LIN {X 0,Y 260.997,Z 552.106,A -85,B 0,C 180,E1 -19941.733,E2 -19941.733} C_VEL
LIN {X 0,Y 261.38,Z 553.874,A -85,B 0,C 180,E1 -19943.77,E2 -19943.77} C_VEL
LIN {X 0,Y 261.439,Z 557.559,A -85,B 0,C 180,E1 -19946.444,E2 -19946.444} C_VEL
LIN {X 0,Y 260.966,Z 561.356,A -85,B 0,C 180,E1 -19948.526,E2 -19948.526} C_VEL
LIN {X 0,Y 260.147,Z 563.053,A -85,B 0,C 180,E1 -19949.117,E2 -19949.117} C_VEL
LIN {X 0,Y 253.93,Z 571.512,A -85,B 0,C 180,E1 -19951.483,E2 -19951.483} C_VEL
LIN {X 0,Y 248.241,Z 578.441,A -85,B 0,C 180,E1 -19953.971,E2 -19953.971} C_VEL
LIN {X 0,Y 243.866,Z 583.268,A -85,B 0,C 180,E1 -19956.205,E2 -19956.205} C_VEL
LIN {X 0,Y 238.865,Z 588.279,A -85,B 0,C 180,E1 -19959.325,E2 -19959.325} C_VEL
LIN {X 0,Y 234.733,Z 591.746,A -85,B 0,C 180,E1 -19962.578,E2 -19962.578} C_VEL
LIN {X 0,Y 232.898,Z 592.963,A -85,B 0,C 180,E1 -19964.242,E2 -19964.242} C_VEL
LIN {X 0,Y 230.123,Z 594.324,A -85,B 0,C 180,E1 -19967.656,E2 -19967.656} C_VEL
LIN {X 0,Y 227.905,Z 594.264,A -85,B 0,C 180,E1 -19971.131,E2 -19971.131} C_VEL
LIN {X 0,Y 226.815,Z 592.766,A -85,B 0,C 180,E1 -19974.667,E2 -19974.667} C_VEL
LIN {X 0,Y 226.415,Z 591.482,A -85,B 0,C 180,E1 -19976.441,E2 -19976.441} C_VEL
LIN {X 0,Y 225.975,Z 587.71,A -85,B 0,C 180,E1 -19980,E2 -19980} C_VEL
LIN {X 0,Y 226.019,Z 583.819,A -85,B 0,C 180,E1 -19982.674,E2 -19982.674} C_VEL
LIN {X 0,Y 226.077,Z 578.823,A -85,B 0,C 180,E1 -19985.352,E2 -19985.352} C_VEL
LIN {X 0,Y 226.623,Z 571.523,A -85,B 0,C 180,E1 -19988.471,E2 -19988.471} C_VEL
LIN {X 0,Y 227.3,Z 563.747,A -85,B 0,C 180,E1 -19991.143,E2 -19991.143} C_VEL
LIN {X 0,Y 228.271,Z 554.253,A -85,B 0,C 180,E1 -19993.805,E2 -19993.805} C_VEL
LIN {X 0,Y 229.552,Z 543.626,A -85,B 0,C 180,E1 -19996.223,E2 -19996.223} C_VEL
LIN {X 0,Y 230.932,Z 531.732,A -85,B 0,C 180,E1 -19998.406,E2 -19998.406} C_VEL
LIN {X 0,Y 232.043,Z 520.197,A -85,B 0,C 180,E1 -20000.13,E2 -20000.13} C_VEL
LIN {X 0,Y 229.504,Z 506.12,A -85,B 0,C 180,E1 -20001.897,E2 -20001.897} C_VEL
LIN {X 0,Y 227.192,Z 492.741,A -85,B 0,C 180,E1 -20003.213,E2 -20003.213} C_VEL
LIN {X 0,Y 226.512,Z 488.275,A -85,B 0,C 180,E1 -20003.585,E2 -20003.585} C_VEL
LIN {X 0,Y 226.901,Z 488.225,A -85,B 0,C 180,E1 -20007.685,E2 -20007.685} C_VEL
LIN {X 0,Y 227.309,Z 488.167,A -85,B 0,C 180,E1 -20011.71,E2 -20011.71} C_VEL
LIN {X 0,Y 227.697,Z 488.121,A -85,B 0,C 180,E1 -20015.906,E2 -20015.906} C_VEL
LIN {X 0,Y 227.817,Z 488.105,A -85,B 0,C 180,E1 -20019.535,E2 -20019.535} C_VEL
LIN {X 0,Y 227.812,Z 488.105,A -85,B 0,C 180,E1 -20022.743,E2 -20022.743} C_VEL
LIN {X 0,Y 227.817,Z 488.105,A -85,B 0,C 180,E1 -20027.259,E2 -20027.259} C_VEL
LIN {X 0,Y 227.873,Z 488.098,A -85,B 0,C 180,E1 -20031.914,E2 -20031.914} C_VEL
LIN {X 0,Y 227.895,Z 488.097,A -85,B 0,C 180,E1 -20036.373,E2 -20036.373} C_VEL
LIN {X 0,Y 227.922,Z 488.093,A -85,B 0,C 180,E1 -20040.438,E2 -20040.438} C_VEL
LIN {X 0,Y 227.933,Z 488.092,A -85,B 0,C 180,E1 -20044.426,E2 -20044.426} C_VEL
LIN {X 0,Y 227.966,Z 488.087,A -85,B 0,C 180,E1 -20048.287,E2 -20048.287} C_VEL
LIN {X 0,Y 228.039,Z 488.078,A -85,B 0,C 180,E1 -20052.826,E2 -20052.826} C_VEL
LIN {X 0,Y 228.099,Z 488.068,A -85,B 0,C 180,E1 -20057.545,E2 -20057.545} C_VEL
LIN {X 0,Y 228.33,Z 488.041,A -85,B 0,C 180,E1 -20061.147,E2 -20061.147} C_VEL
LIN {X 0,Y 228.363,Z 488.036,A -85,B 0,C 180,E1 -20062.929,E2 -20062.929} C_VEL
LIN {X 0,Y 228.559,Z 488.015,A -85,B 0,C 180,E1 -20068.238,E2 -20068.238} C_VEL
LIN {X 0,Y 228.558,Z 488.015,A -85,B 0,C 180,E1 -20071.762,E2 -20071.762} C_VEL
LIN {X 0,Y 228.316,Z 488.042,A -85,B 0,C 180,E1 -20077.073,E2 -20077.073} C_VEL
LIN {X 0,Y 228.15,Z 488.063,A -85,B 0,C 180,E1 -20080.651,E2 -20080.651} C_VEL
LIN {X 0,Y 228.07,Z 488.074,A -85,B 0,C 180,E1 -20084.272,E2 -20084.272} C_VEL
LIN {X 0,Y 228.007,Z 488.085,A -85,B 0,C 180,E1 -20087.953,E2 -20087.953} C_VEL
LIN {X 0,Y 227.934,Z 488.089,A -85,B 0,C 180,E1 -20092.329,E2 -20092.329} C_VEL
LIN {X 0,Y 227.947,Z 488.089,A -85,B 0,C 180,E1 -20096.602,E2 -20096.602} C_VEL
LIN {X 0,Y 227.912,Z 488.091,A -85,B 0,C 180,E1 -20100.296,E2 -20100.296} C_VEL
LIN {X 0,Y 227.894,Z 488.098,A -85,B 0,C 180,E1 -20103.718,E2 -20103.718} C_VEL
LIN {X 0,Y 227.873,Z 488.098,A -85,B 0,C 180,E1 -20108.086,E2 -20108.086} C_VEL
LIN {X 0,Y 227.817,Z 488.105,A -85,B 0,C 180,E1 -20112.741,E2 -20112.741} C_VEL
LIN {X 0,Y 227.814,Z 488.105,A -85,B 0,C 180,E1 -20117.257,E2 -20117.257} C_VEL
LIN {X 0,Y 227.826,Z 488.107,A -85,B 0,C 180,E1 -20121.905,E2 -20121.905} C_VEL
LIN {X 0,Y 227.775,Z 488.111,A -85,B 0,C 180,E1 -20124.108,E2 -20124.108} C_VEL
LIN {X 0,Y 227.441,Z 488.151,A -85,B 0,C 180,E1 -20128.31,E2 -20128.31} C_VEL
LIN {X 0,Y 226.941,Z 488.214,A -85,B 0,C 180,E1 -20132.32,E2 -20132.32} C_VEL
LIN {X 0,Y 226.511,Z 488.447,A -85,B 0,C 180,E1 -20136.724,E2 -20136.724} C_VEL
LIN {X 0,Y 228.847,Z 502.265,A -85,B 0,C 180,E1 -20137.982,E2 -20137.982} C_VEL
LIN {X 0,Y 231.402,Z 516.968,A -85,B 0,C 180,E1 -20139.723,E2 -20139.723} C_VEL
LIN {X 0,Y 231.9,Z 519.763,A -85,B 0,C 180,E1 -20140.109,E2 -20140.109} C_VEL
LIN {X 0,Y 230.711,Z 532.571,A -85,B 0,C 180,E1 -20142.035,E2 -20142.035} C_VEL
LIN {X 0,Y 229.325,Z 544.216,A -85,B 0,C 180,E1 -20144.217,E2 -20144.217} C_VEL
LIN {X 0,Y 228.097,Z 554.659,A -85,B 0,C 180,E1 -20146.638,E2 -20146.638} C_VEL
LIN {X 0,Y 227.17,Z 564.012,A -85,B 0,C 180,E1 -20149.302,E2 -20149.302} C_VEL
LIN {X 0,Y 226.478,Z 571.65,A -85,B 0,C 180,E1 -20151.972,E2 -20151.972} C_VEL
LIN {X 0,Y 226.06,Z 577.897,A -85,B 0,C 180,E1 -20154.648,E2 -20154.648} C_VEL
LIN {X 0,Y 226.009,Z 582.973,A -85,B 0,C 180,E1 -20157.326,E2 -20157.326} C_VEL
LIN {X 0,Y 225.947,Z 586.927,A -85,B 0,C 180,E1 -20160,E2 -20160} C_VEL
LIN {X 0,Y 226.391,Z 590.762,A -85,B 0,C 180,E1 -20163.559,E2 -20163.559} C_VEL
LIN {X 0,Y 227.153,Z 593.019,A -85,B 0,C 180,E1 -20167.109,E2 -20167.109} C_VEL
LIN {X 0,Y 228.816,Z 593.825,A -85,B 0,C 180,E1 -20170.619,E2 -20170.619} C_VEL
LIN {X 0,Y 229.985,Z 593.691,A -85,B 0,C 180,E1 -20172.351,E2 -20172.351} C_VEL
LIN {X 0,Y 231.149,Z 593.198,A -85,B 0,C 180,E1 -20174.077,E2 -20174.077} C_VEL
LIN {X 0,Y 234.587,Z 591.116,A -85,B 0,C 180,E1 -20177.433,E2 -20177.433} C_VEL
LIN {X 0,Y 236.432,Z 589.575,A -85,B 0,C 180,E1 -20179.085,E2 -20179.085} C_VEL
LIN {X 0,Y 241.087,Z 585.314,A -85,B 0,C 180,E1 -20182.269,E2 -20182.269} C_VEL
LIN {X 0,Y 246.476,Z 579.492,A -85,B 0,C 180,E1 -20185.322,E2 -20185.322} C_VEL
LIN {X 0,Y 251.935,Z 572.921,A -85,B 0,C 180,E1 -20187.856,E2 -20187.856} C_VEL
LIN {X 0,Y 257.976,Z 564.873,A -85,B 0,C 180,E1 -20190.264,E2 -20190.264} C_VEL
LIN {X 0,Y 261.362,Z 559.796,A -85,B 0,C 180,E1 -20191.544,E2 -20191.544} C_VEL
LIN {X 0,Y 262.125,Z 555.274,A -85,B 0,C 180,E1 -20193.782,E2 -20193.782} C_VEL
LIN {X 0,Y 262.421,Z 551.482,A -85,B 0,C 180,E1 -20196.099,E2 -20196.099} C_VEL
LIN {X 0,Y 262.376,Z 549.202,A -85,B 0,C 180,E1 -20198.03,E2 -20198.03} C_VEL
LIN {X 0,Y 262.053,Z 547.219,A -85,B 0,C 180,E1 -20201.329,E2 -20201.329} C_VEL
LIN {X 0,Y 262.112,Z 546.874,A -85,B 0,C 180,E1 -20204.198,E2 -20204.198} C_VEL
LIN {X 0,Y 262.067,Z 548.078,A -85,B 0,C 180,E1 -20206.392,E2 -20206.392} C_VEL
LIN {X 0,Y 262.09,Z 550.434,A -85,B 0,C 180,E1 -20208.662,E2 -20208.662} C_VEL
LIN {X 0,Y 261.725,Z 553.395,A -85,B 0,C 180,E1 -20210.385,E2 -20210.385} C_VEL
LIN {X 0,Y 261.022,Z 556.614,A -85,B 0,C 180,E1 -20211.737,E2 -20211.737} C_VEL
LIN {X 0,Y 259.769,Z 560.538,A -85,B 0,C 180,E1 -20213.058,E2 -20213.058} C_VEL
LIN {X 0,Y 258.835,Z 562.899,A -85,B 0,C 180,E1 -20213.731,E2 -20213.731} C_VEL
LIN {X 0,Y 256.688,Z 566.806,A -85,B 0,C 180,E1 -20214.61,E2 -20214.61} C_VEL
LIN {X 0,Y 250.235,Z 576.094,A -85,B 0,C 180,E1 -20216.484,E2 -20216.484} C_VEL
LIN {X 0,Y 247.787,Z 579.695,A -85,B 0,C 180,E1 -20217.424,E2 -20217.424} C_VEL
LIN {X 0,Y 247.137,Z 580.788,A -85,B 0,C 180,E1 -20217.775,E2 -20217.775} C_VEL
LIN {X 0,Y 242.575,Z 587.784,A -85,B 0,C 180,E1 -20220.015,E2 -20220.015} C_VEL
LIN {X 0,Y 236.889,Z 595.016,A -85,B 0,C 180,E1 -20222.622,E2 -20222.622} C_VEL
LIN {X 0,Y 231.389,Z 601.575,A -85,B 0,C 180,E1 -20225.697,E2 -20225.697} C_VEL
LIN {X 0,Y 227.708,Z 605.755,A -85,B 0,C 180,E1 -20228.262,E2 -20228.262} C_VEL
LIN {X 0,Y 224.049,Z 609.838,A -85,B 0,C 180,E1 -20231.719,E2 -20231.719} C_VEL
LIN {X 0,Y 221.143,Z 612.568,A -85,B 0,C 180,E1 -20235.271,E2 -20235.271} C_VEL
LIN {X 0,Y 219.574,Z 613.972,A -85,B 0,C 180,E1 -20238.928,E2 -20238.928} C_VEL
LIN {X 0,Y 218.936,Z 613.961,A -85,B 0,C 180,E1 -20242.623,E2 -20242.623} C_VEL
LIN {X 0,Y 218.988,Z 612.5,A -85,B 0,C 180,E1 -20246.32,E2 -20246.32} C_VEL
LIN {X 0,Y 219.639,Z 610.27,A -85,B 0,C 180,E1 -20249.312,E2 -20249.312} C_VEL
LIN {X 0,Y 219.273,Z 612.678,A -85,B 0,C 180,E1 -20251.837,E2 -20251.837} C_VEL
LIN {X 0,Y 218.885,Z 614.828,A -85,B 0,C 180,E1 -20255.528,E2 -20255.528} C_VEL
LIN {X 0,Y 219.122,Z 615.516,A -85,B 0,C 180,E1 -20259.228,E2 -20259.228} C_VEL
LIN {X 0,Y 220.226,Z 614.78,A -85,B 0,C 180,E1 -20262.908,E2 -20262.908} C_VEL
LIN {X 0,Y 222.43,Z 612.714,A -85,B 0,C 180,E1 -20266.521,E2 -20266.521} C_VEL
LIN {X 0,Y 225.697,Z 609.304,A -85,B 0,C 180,E1 -20270.031,E2 -20270.031} C_VEL
LIN {X 0,Y 228.769,Z 605.775,A -85,B 0,C 180,E1 -20272.65,E2 -20272.65} C_VEL
LIN {X 0,Y 233.83,Z 599.998,A -85,B 0,C 180,E1 -20275.837,E2 -20275.837} C_VEL
LIN {X 0,Y 239.21,Z 593.581,A -85,B 0,C 180,E1 -20278.518,E2 -20278.518} C_VEL
LIN {X 0,Y 245.963,Z 584.688,A -85,B 0,C 180,E1 -20281.431,E2 -20281.431} C_VEL
LIN {X 0,Y 248.001,Z 581.154,A -85,B 0,C 180,E1 -20282.577,E2 -20282.577} C_VEL
LIN {X 0,Y 250.573,Z 575.348,A -85,B 0,C 180,E1 -20284.659,E2 -20284.659} C_VEL
LIN {X 0,Y 252.859,Z 568.813,A -85,B 0,C 180,E1 -20287.194,E2 -20287.194} C_VEL
LIN {X 0,Y 254.372,Z 563.772,A -85,B 0,C 180,E1 -20289.455,E2 -20289.455} C_VEL
LIN {X 0,Y 255.197,Z 560.413,A -85,B 0,C 180,E1 -20291.372,E2 -20291.372} C_VEL
LIN {X 0,Y 255.721,Z 557.205,A -85,B 0,C 180,E1 -20294.393,E2 -20294.393} C_VEL
LIN {X 0,Y 255.885,Z 556.408,A -85,B 0,C 180,E1 -20295.57,E2 -20295.57} C_VEL
LIN {X 0,Y 255.914,Z 556.069,A -85,B 0,C 180,E1 -20297.858,E2 -20297.858} C_VEL
LIN {X 0,Y 256.096,Z 556.949,A -85,B 0,C 180,E1 -20300.863,E2 -20300.863} C_VEL
LIN {X 0,Y 256.423,Z 559.105,A -85,B 0,C 180,E1 -20303.785,E2 -20303.785} C_VEL
LIN {X 0,Y 256.219,Z 561.054,A -85,B 0,C 180,E1 -20305.375,E2 -20305.375} C_VEL
LIN {X 0,Y 255.687,Z 564.505,A -85,B 0,C 180,E1 -20307.604,E2 -20307.604} C_VEL
LIN {X 0,Y 254.559,Z 566.477,A -85,B 0,C 180,E1 -20308.362,E2 -20308.362} C_VEL
LIN {X 0,Y 248.996,Z 573.361,A -85,B 0,C 180,E1 -20310.4,E2 -20310.4} C_VEL
LIN {X 0,Y 242.182,Z 580.837,A -85,B 0,C 180,E1 -20313.269,E2 -20313.269} C_VEL
LIN {X 0,Y 237.648,Z 585.3,A -85,B 0,C 180,E1 -20315.542,E2 -20315.542} C_VEL
LIN {X 0,Y 232.423,Z 589.852,A -85,B 0,C 180,E1 -20318.725,E2 -20318.725} C_VEL
LIN {X 0,Y 228.076,Z 592.969,A -85,B 0,C 180,E1 -20322.053,E2 -20322.053} C_VEL
LIN {X 0,Y 226.163,Z 594.008,A -85,B 0,C 180,E1 -20323.76,E2 -20323.76} C_VEL
LIN {X 0,Y 223.23,Z 595.007,A -85,B 0,C 180,E1 -20327.269,E2 -20327.269} C_VEL
LIN {X 0,Y 220.918,Z 594.665,A -85,B 0,C 180,E1 -20330.848,E2 -20330.848} C_VEL
LIN {X 0,Y 219.753,Z 592.868,A -85,B 0,C 180,E1 -20334.495,E2 -20334.495} C_VEL
LIN {X 0,Y 219.051,Z 589.599,A -85,B 0,C 180,E1 -20338.162,E2 -20338.162} C_VEL
LIN {X 0,Y 218.882,Z 586.103,A -85,B 0,C 180,E1 -20340.92,E2 -20340.92} C_VEL
LIN {X 0,Y 218.927,Z 581.625,A -85,B 0,C 180,E1 -20343.682,E2 -20343.682} C_VEL
LIN {X 0,Y 219.255,Z 575.022,A -85,B 0,C 180,E1 -20346.904,E2 -20346.904} C_VEL
LIN {X 0,Y 219.77,Z 567.895,A -85,B 0,C 180,E1 -20349.666,E2 -20349.666} C_VEL
LIN {X 0,Y 220.638,Z 559.205,A -85,B 0,C 180,E1 -20352.417,E2 -20352.417} C_VEL
LIN {X 0,Y 221.801,Z 548.639,A -85,B 0,C 180,E1 -20355.154,E2 -20355.154} C_VEL
LIN {X 0,Y 223.055,Z 537.863,A -85,B 0,C 180,E1 -20357.418,E2 -20357.418} C_VEL
LIN {X 0,Y 224.214,Z 527.533,A -85,B 0,C 180,E1 -20359.216,E2 -20359.216} C_VEL
LIN {X 0,Y 224.919,Z 521.594,A -85,B 0,C 180,E1 -20360.104,E2 -20360.104} C_VEL
LIN {X 0,Y 223.269,Z 511.586,A -85,B 0,C 180,E1 -20361.465,E2 -20361.465} C_VEL
LIN {X 0,Y 220.895,Z 498.112,A -85,B 0,C 180,E1 -20362.962,E2 -20362.962} C_VEL
LIN {X 0,Y 219.504,Z 489.148,A -85,B 0,C 180,E1 -20363.777,E2 -20363.777} C_VEL
LIN {X 0,Y 219.95,Z 489.087,A -85,B 0,C 180,E1 -20368.64,E2 -20368.64} C_VEL
LIN {X 0,Y 220.361,Z 489.032,A -85,B 0,C 180,E1 -20372.833,E2 -20372.833} C_VEL
LIN {X 0,Y 220.71,Z 488.99,A -85,B 0,C 180,E1 -20377.243,E2 -20377.243} C_VEL
LIN {X 0,Y 220.776,Z 488.984,A -85,B 0,C 180,E1 -20380.182,E2 -20380.182} C_VEL
LIN {X 0,Y 220.776,Z 488.985,A -85,B 0,C 180,E1 -20384.454,E2 -20384.454} C_VEL
LIN {X 0,Y 220.778,Z 488.984,A -85,B 0,C 180,E1 -20388.049,E2 -20388.049} C_VEL
LIN {X 0,Y 220.835,Z 488.975,A -85,B 0,C 180,E1 -20392.795,E2 -20392.795} C_VEL
LIN {X 0,Y 220.828,Z 488.975,A -85,B 0,C 180,E1 -20397.246,E2 -20397.246} C_VEL
LIN {X 0,Y 220.84,Z 488.973,A -85,B 0,C 180,E1 -20401.487,E2 -20401.487} C_VEL
LIN {X 0,Y 220.871,Z 488.971,A -85,B 0,C 180,E1 -20405.565,E2 -20405.565} C_VEL
LIN {X 0,Y 220.897,Z 488.965,A -85,B 0,C 180,E1 -20409.514,E2 -20409.514} C_VEL
LIN {X 0,Y 221.021,Z 488.952,A -85,B 0,C 180,E1 -20413.37,E2 -20413.37} C_VEL
LIN {X 0,Y 221.121,Z 488.938,A -85,B 0,C 180,E1 -20419.006,E2 -20419.006} C_VEL
LIN {X 0,Y 221.316,Z 488.915,A -85,B 0,C 180,E1 -20422.702,E2 -20422.702} C_VEL
LIN {X 0,Y 221.517,Z 488.893,A -85,B 0,C 180,E1 -20428.182,E2 -20428.182} C_VEL
LIN {X 0,Y 221.516,Z 488.893,A -85,B 0,C 180,E1 -20431.818,E2 -20431.818} C_VEL
LIN {X 0,Y 221.252,Z 488.923,A -85,B 0,C 180,E1 -20437.3,E2 -20437.3} C_VEL
LIN {X 0,Y 221.086,Z 488.943,A -85,B 0,C 180,E1 -20440.996,E2 -20440.996} C_VEL
LIN {X 0,Y 221.021,Z 488.952,A -85,B 0,C 180,E1 -20446.63,E2 -20446.63} C_VEL
LIN {X 0,Y 220.897,Z 488.966,A -85,B 0,C 180,E1 -20450.486,E2 -20450.486} C_VEL
LIN {X 0,Y 220.871,Z 488.971,A -85,B 0,C 180,E1 -20454.435,E2 -20454.435} C_VEL
LIN {X 0,Y 220.84,Z 488.973,A -85,B 0,C 180,E1 -20458.513,E2 -20458.513} C_VEL
LIN {X 0,Y 220.828,Z 488.975,A -85,B 0,C 180,E1 -20462.754,E2 -20462.754} C_VEL
LIN {X 0,Y 220.842,Z 488.974,A -85,B 0,C 180,E1 -20467.288,E2 -20467.288} C_VEL
LIN {X 0,Y 220.778,Z 488.984,A -85,B 0,C 180,E1 -20471.951,E2 -20471.951} C_VEL
LIN {X 0,Y 220.777,Z 488.985,A -85,B 0,C 180,E1 -20475.546,E2 -20475.546} C_VEL
LIN {X 0,Y 220.79,Z 488.98,A -85,B 0,C 180,E1 -20480.459,E2 -20480.459} C_VEL
LIN {X 0,Y 220.788,Z 488.981,A -85,B 0,C 180,E1 -20482.785,E2 -20482.785} C_VEL
LIN {X 0,Y 220.456,Z 489.02,A -85,B 0,C 180,E1 -20487.183,E2 -20487.183} C_VEL
LIN {X 0,Y 220.268,Z 489.047,A -85,B 0,C 180,E1 -20489.483,E2 -20489.483} C_VEL
LIN {X 0,Y 219.752,Z 489.112,A -85,B 0,C 180,E1 -20493.571,E2 -20493.571} C_VEL
LIN {X 0,Y 219.454,Z 489.149,A -85,B 0,C 180,E1 -20496.505,E2 -20496.505} C_VEL
LIN {X 0,Y 222.105,Z 504.713,A -85,B 0,C 180,E1 -20498.039,E2 -20498.039} C_VEL
LIN {X 0,Y 224.317,Z 517.522,A -85,B 0,C 180,E1 -20499.625,E2 -20499.625} C_VEL
LIN {X 0,Y 224.798,Z 521.395,A -85,B 0,C 180,E1 -20500.176,E2 -20500.176} C_VEL
LIN {X 0,Y 223.456,Z 533.723,A -85,B 0,C 180,E1 -20502.142,E2 -20502.142} C_VEL
LIN {X 0,Y 222.089,Z 545.146,A -85,B 0,C 180,E1 -20504.396,E2 -20504.396} C_VEL
LIN {X 0,Y 220.841,Z 556.293,A -85,B 0,C 180,E1 -20507.128,E2 -20507.128} C_VEL
LIN {X 0,Y 219.895,Z 565.419,A -85,B 0,C 180,E1 -20509.875,E2 -20509.875} C_VEL
LIN {X 0,Y 219.311,Z 572.892,A -85,B 0,C 180,E1 -20512.635,E2 -20512.635} C_VEL
LIN {X 0,Y 218.945,Z 579.457,A -85,B 0,C 180,E1 -20515.643,E2 -20515.643} C_VEL
LIN {X 0,Y 218.9,Z 583.873,A -85,B 0,C 180,E1 -20518.16,E2 -20518.16} C_VEL
LIN {X 0,Y 218.918,Z 587.74,A -85,B 0,C 180,E1 -20520.919,E2 -20520.919} C_VEL
LIN {X 0,Y 219.332,Z 590.677,A -85,B 0,C 180,E1 -20523.674,E2 -20523.674} C_VEL
LIN {X 0,Y 220.113,Z 593.248,A -85,B 0,C 180,E1 -20527.337,E2 -20527.337} C_VEL
LIN {X 0,Y 221.875,Z 594.342,A -85,B 0,C 180,E1 -20530.955,E2 -20530.955} C_VEL
LIN {X 0,Y 224.34,Z 594.036,A -85,B 0,C 180,E1 -20534.514,E2 -20534.514} C_VEL
LIN {X 0,Y 225.965,Z 593.365,A -85,B 0,C 180,E1 -20536.255,E2 -20536.255} C_VEL
LIN {X 0,Y 229.887,Z 590.951,A -85,B 0,C 180,E1 -20539.65,E2 -20539.65} C_VEL
LIN {X 0,Y 234.75,Z 587.071,A -85,B 0,C 180,E1 -20542.904,E2 -20542.904} C_VEL
LIN {X 0,Y 238.859,Z 583.221,A -85,B 0,C 180,E1 -20545.254,E2 -20545.254} C_VEL
LIN {X 0,Y 245.201,Z 576.599,A -85,B 0,C 180,E1 -20548.224,E2 -20548.224} C_VEL
LIN {X 0,Y 251.402,Z 569.264,A -85,B 0,C 180,E1 -20550.676,E2 -20550.676} C_VEL
LIN {X 0,Y 256.107,Z 563.154,A -85,B 0,C 180,E1 -20552.351,E2 -20552.351} C_VEL
LIN {X 0,Y 256.842,Z 560.292,A -85,B 0,C 180,E1 -20553.879,E2 -20553.879} C_VEL
LIN {X 0,Y 257.63,Z 555.851,A -85,B 0,C 180,E1 -20556.88,E2 -20556.88} C_VEL
LIN {X 0,Y 257.614,Z 554.045,A -85,B 0,C 180,E1 -20558.863,E2 -20558.863} C_VEL
LIN {X 0,Y 257.573,Z 552.939,A -85,B 0,C 180,E1 -20560.908,E2 -20560.908} C_VEL
LIN {X 0,Y 257.643,Z 552.453,A -85,B 0,C 180,E1 -20562.996,E2 -20562.996} C_VEL
LIN {X 0,Y 257.679,Z 552.943,A -85,B 0,C 180,E1 -20565.164,E2 -20565.164} C_VEL
LIN {X 0,Y 257.575,Z 554.708,A -85,B 0,C 180,E1 -20567.451,E2 -20567.451} C_VEL
LIN {X 0,Y 257.335,Z 556.746,A -85,B 0,C 180,E1 -20569.046,E2 -20569.046} C_VEL
LIN {X 0,Y 256.636,Z 559.345,A -85,B 0,C 180,E1 -20570.422,E2 -20570.422} C_VEL
LIN {X 0,Y 255.073,Z 563.625,A -85,B 0,C 180,E1 -20572.061,E2 -20572.061} C_VEL
LIN {X 0,Y 251.472,Z 572.097,A -85,B 0,C 180,E1 -20574.936,E2 -20574.936} C_VEL
LIN {X 0,Y 247.137,Z 580.788,A -85,B 0,C 180,E1 -20577.775,E2 -20577.775} C_VEL
LIN {X 0,Y 245.627,Z 583.103,A -85,B 0,C 180,E1 -20578.447,E2 -20578.447} C_VEL
LIN {X 0,Y 243.607,Z 585.428,A -85,B 0,C 180,E1 -20579.031,E2 -20579.031} C_VEL
LIN {X 0,Y 238.671,Z 589.999,A -85,B 0,C 180,E1 -20580.063,E2 -20580.063} C_VEL
LIN {X 0,Y 232.309,Z 595.17,A -85,B 0,C 180,E1 -20581.442,E2 -20581.442} C_VEL
LIN {X 0,Y 229.34,Z 597.864,A -85,B 0,C 180,E1 -20582.513,E2 -20582.513} C_VEL
LIN {X 0,Y 223.497,Z 603.91,A -85,B 0,C 180,E1 -20585.871,E2 -20585.871} C_VEL
LIN {X 0,Y 219.113,Z 608.319,A -85,B 0,C 180,E1 -20589.34,E2 -20589.34} C_VEL
LIN {X 0,Y 215.641,Z 611.397,A -85,B 0,C 180,E1 -20592.943,E2 -20592.943} C_VEL
LIN {X 0,Y 213.263,Z 613.115,A -85,B 0,C 180,E1 -20596.663,E2 -20596.663} C_VEL
LIN {X 0,Y 212.112,Z 613.505,A -85,B 0,C 180,E1 -20600.464,E2 -20600.464} C_VEL
LIN {X 0,Y 211.891,Z 612.547,A -85,B 0,C 180,E1 -20604.289,E2 -20604.289} C_VEL
LIN {X 0,Y 212.355,Z 610.087,A -85,B 0,C 180,E1 -20608.103,E2 -20608.103} C_VEL
LIN {X 0,Y 212.65,Z 609.071,A -85,B 0,C 180,E1 -20609.408,E2 -20609.408} C_VEL
LIN {X 0,Y 212.258,Z 611.558,A -85,B 0,C 180,E1 -20611.897,E2 -20611.897} C_VEL
LIN {X 0,Y 211.848,Z 613.936,A -85,B 0,C 180,E1 -20615.712,E2 -20615.712} C_VEL
LIN {X 0,Y 212.11,Z 614.863,A -85,B 0,C 180,E1 -20619.536,E2 -20619.536} C_VEL
LIN {X 0,Y 213.274,Z 614.442,A -85,B 0,C 180,E1 -20623.337,E2 -20623.337} C_VEL
LIN {X 0,Y 215.63,Z 612.708,A -85,B 0,C 180,E1 -20627.058,E2 -20627.058} C_VEL
LIN {X 0,Y 219.038,Z 609.647,A -85,B 0,C 180,E1 -20630.668,E2 -20630.668} C_VEL
LIN {X 0,Y 223.434,Z 605.247,A -85,B 0,C 180,E1 -20634.136,E2 -20634.136} C_VEL
LIN {X 0,Y 229.053,Z 599.465,A -85,B 0,C 180,E1 -20637.403,E2 -20637.403} C_VEL
LIN {X 0,Y 235.741,Z 592.142,A -85,B 0,C 180,E1 -20640.452,E2 -20640.452} C_VEL
LIN {X 0,Y 240.974,Z 585.649,A -85,B 0,C 180,E1 -20642.653,E2 -20642.653} C_VEL
LIN {X 0,Y 243.592,Z 581.333,A -85,B 0,C 180,E1 -20644.236,E2 -20644.236} C_VEL
LIN {X 0,Y 246.525,Z 575.041,A -85,B 0,C 180,E1 -20646.775,E2 -20646.775} C_VEL
LIN {X 0,Y 248.594,Z 569.983,A -85,B 0,C 180,E1 -20649.03,E2 -20649.03} C_VEL
LIN {X 0,Y 249.912,Z 566.177,A -85,B 0,C 180,E1 -20651.088,E2 -20651.088} C_VEL
LIN {X 0,Y 250.432,Z 564.484,A -85,B 0,C 180,E1 -20652.34,E2 -20652.34} C_VEL
LIN {X 0,Y 250.888,Z 562.482,A -85,B 0,C 180,E1 -20654.452,E2 -20654.452} C_VEL
LIN {X 0,Y 251.089,Z 561.703,A -85,B 0,C 180,E1 -20655.593,E2 -20655.593} C_VEL
LIN {X 0,Y 251.194,Z 561.354,A -85,B 0,C 180,E1 -20656.672,E2 -20656.672} C_VEL
LIN {X 0,Y 251.109,Z 561.756,A -85,B 0,C 180,E1 -20659.93,E2 -20659.93} C_VEL
LIN {X 0,Y 251.188,Z 562.769,A -85,B 0,C 180,E1 -20662.009,E2 -20662.009} C_VEL
LIN {X 0,Y 251.114,Z 564.633,A -85,B 0,C 180,E1 -20664.256,E2 -20664.256} C_VEL
LIN {X 0,Y 250.324,Z 567.979,A -85,B 0,C 180,E1 -20666.806,E2 -20666.806} C_VEL
LIN {X 0,Y 248.986,Z 569.913,A -85,B 0,C 180,E1 -20667.568,E2 -20667.568} C_VEL
LIN {X 0,Y 241.404,Z 578.164,A -85,B 0,C 180,E1 -20670.336,E2 -20670.336} C_VEL
LIN {X 0,Y 236.157,Z 583.178,A -85,B 0,C 180,E1 -20672.531,E2 -20672.531} C_VEL
LIN {X 0,Y 230.027,Z 588.425,A -85,B 0,C 180,E1 -20675.641,E2 -20675.641} C_VEL
LIN {X 0,Y 225.979,Z 591.397,A -85,B 0,C 180,E1 -20678.087,E2 -20678.087} C_VEL
LIN {X 0,Y 221.429,Z 594.12,A -85,B 0,C 180,E1 -20681.495,E2 -20681.495} C_VEL
LIN {X 0,Y 217.797,Z 595.488,A -85,B 0,C 180,E1 -20685.04,E2 -20685.04} C_VEL
LIN {X 0,Y 214.98,Z 595.507,A -85,B 0,C 180,E1 -20688.689,E2 -20688.689} C_VEL
LIN {X 0,Y 213.192,Z 594.104,A -85,B 0,C 180,E1 -20692.423,E2 -20692.423} C_VEL
LIN {X 0,Y 212.3,Z 591.302,A -85,B 0,C 180,E1 -20696.204,E2 -20696.204} C_VEL
LIN {X 0,Y 211.878,Z 588.198,A -85,B 0,C 180,E1 -20699.05,E2 -20699.05} C_VEL
LIN {X 0,Y 211.852,Z 584.159,A -85,B 0,C 180,E1 -20701.902,E2 -20701.902} C_VEL
LIN {X 0,Y 211.918,Z 578.53,A -85,B 0,C 180,E1 -20705.024,E2 -20705.024} C_VEL
LIN {X 0,Y 212.393,Z 571.648,A -85,B 0,C 180,E1 -20708.085,E2 -20708.085} C_VEL
LIN {X 0,Y 213.192,Z 562.296,A -85,B 0,C 180,E1 -20711.408,E2 -20711.408} C_VEL
LIN {X 0,Y 214.047,Z 554.112,A -85,B 0,C 180,E1 -20713.772,E2 -20713.772} C_VEL
LIN {X 0,Y 215.369,Z 543.318,A -85,B 0,C 180,E1 -20716.348,E2 -20716.348} C_VEL
LIN {X 0,Y 216.798,Z 531.37,A -85,B 0,C 180,E1 -20718.671,E2 -20718.671} C_VEL
LIN {X 0,Y 217.782,Z 520.974,A -85,B 0,C 180,E1 -20720.321,E2 -20720.321} C_VEL
LIN {X 0,Y 215.329,Z 507.306,A -85,B 0,C 180,E1 -20722.153,E2 -20722.153} C_VEL
LIN {X 0,Y 213.102,Z 494.095,A -85,B 0,C 180,E1 -20723.553,E2 -20723.553} C_VEL
LIN {X 0,Y 212.469,Z 490.024,A -85,B 0,C 180,E1 -20723.969,E2 -20723.969} C_VEL
LIN {X 0,Y 212.754,Z 489.987,A -85,B 0,C 180,E1 -20727.547,E2 -20727.547} C_VEL
LIN {X 0,Y 213.205,Z 489.925,A -85,B 0,C 180,E1 -20731.832,E2 -20731.832} C_VEL
LIN {X 0,Y 213.503,Z 489.889,A -85,B 0,C 180,E1 -20734.619,E2 -20734.619} C_VEL
LIN {X 0,Y 213.667,Z 489.868,A -85,B 0,C 180,E1 -20738.68,E2 -20738.68} C_VEL
LIN {X 0,Y 213.707,Z 489.859,A -85,B 0,C 180,E1 -20741.127,E2 -20741.127} C_VEL
LIN {X 0,Y 213.708,Z 489.862,A -85,B 0,C 180,E1 -20743.679,E2 -20743.679} C_VEL
LIN {X 0,Y 213.711,Z 489.865,A -85,B 0,C 180,E1 -20746.344,E2 -20746.344} C_VEL
LIN {X 0,Y 213.739,Z 489.856,A -85,B 0,C 180,E1 -20751.336,E2 -20751.336} C_VEL
LIN {X 0,Y 213.774,Z 489.857,A -85,B 0,C 180,E1 -20756.021,E2 -20756.021} C_VEL
LIN {X 0,Y 213.784,Z 489.854,A -85,B 0,C 180,E1 -20760.454,E2 -20760.454} C_VEL
LIN {X 0,Y 213.806,Z 489.851,A -85,B 0,C 180,E1 -20764.702,E2 -20764.702} C_VEL
LIN {X 0,Y 213.817,Z 489.847,A -85,B 0,C 180,E1 -20768.804,E2 -20768.804} C_VEL
LIN {X 0,Y 213.948,Z 489.833,A -85,B 0,C 180,E1 -20772.804,E2 -20772.804} C_VEL
LIN {X 0,Y 213.985,Z 489.825,A -85,B 0,C 180,E1 -20776.709,E2 -20776.709} C_VEL
LIN {X 0,Y 214.201,Z 489.802,A -85,B 0,C 180,E1 -20780.558,E2 -20780.558} C_VEL
LIN {X 0,Y 214.253,Z 489.795,A -85,B 0,C 180,E1 -20782.46,E2 -20782.46} C_VEL
LIN {X 0,Y 214.451,Z 489.773,A -85,B 0,C 180,E1 -20788.122,E2 -20788.122} C_VEL
LIN {X 0,Y 214.555,Z 489.761,A -85,B 0,C 180,E1 -20790,E2 -20790} C_VEL
LIN {X 0,Y 214.448,Z 489.773,A -85,B 0,C 180,E1 -20791.878,E2 -20791.878} C_VEL
LIN {X 0,Y 214.193,Z 489.803,A -85,B 0,C 180,E1 -20797.542,E2 -20797.542} C_VEL
LIN {X 0,Y 214.012,Z 489.825,A -85,B 0,C 180,E1 -20801.364,E2 -20801.364} C_VEL
LIN {X 0,Y 213.938,Z 489.833,A -85,B 0,C 180,E1 -20805.237,E2 -20805.237} C_VEL
LIN {X 0,Y 213.844,Z 489.846,A -85,B 0,C 180,E1 -20809.187,E2 -20809.187} C_VEL
LIN {X 0,Y 213.851,Z 489.843,A -85,B 0,C 180,E1 -20813.227,E2 -20813.227} C_VEL
LIN {X 0,Y 213.833,Z 489.849,A -85,B 0,C 180,E1 -20817.45,E2 -20817.45} C_VEL
LIN {X 0,Y 213.783,Z 489.853,A -85,B 0,C 180,E1 -20821.735,E2 -20821.735} C_VEL
LIN {X 0,Y 213.756,Z 489.857,A -85,B 0,C 180,E1 -20826.286,E2 -20826.286} C_VEL
LIN {X 0,Y 213.719,Z 489.86,A -85,B 0,C 180,E1 -20831.124,E2 -20831.124} C_VEL
LIN {X 0,Y 213.711,Z 489.866,A -85,B 0,C 180,E1 -20833.678,E2 -20833.678} C_VEL
LIN {X 0,Y 213.709,Z 489.861,A -85,B 0,C 180,E1 -20836.344,E2 -20836.344} C_VEL
LIN {X 0,Y 213.715,Z 489.859,A -85,B 0,C 180,E1 -20839.144,E2 -20839.144} C_VEL
LIN {X 0,Y 213.664,Z 489.871,A -85,B 0,C 180,E1 -20843.695,E2 -20843.695} C_VEL
LIN {X 0,Y 213.522,Z 489.884,A -85,B 0,C 180,E1 -20845.975,E2 -20845.975} C_VEL
LIN {X 0,Y 213.068,Z 489.943,A -85,B 0,C 180,E1 -20850.345,E2 -20850.345} C_VEL
LIN {X 0,Y 212.497,Z 490.014,A -85,B 0,C 180,E1 -20855.58,E2 -20855.58} C_VEL
LIN {X 0,Y 212.432,Z 490.023,A -85,B 0,C 180,E1 -20856.382,E2 -20856.382} C_VEL
LIN {X 0,Y 214.965,Z 505.131,A -85,B 0,C 180,E1 -20857.917,E2 -20857.917} C_VEL
LIN {X 0,Y 217.341,Z 518.757,A -85,B 0,C 180,E1 -20859.678,E2 -20859.678} C_VEL
LIN {X 0,Y 217.74,Z 521.066,A -85,B 0,C 180,E1 -20860.02,E2 -20860.02} C_VEL
LIN {X 0,Y 216.387,Z 533.416,A -85,B 0,C 180,E1 -20862.028,E2 -20862.028} C_VEL
LIN {X 0,Y 214.977,Z 544.933,A -85,B 0,C 180,E1 -20864.353,E2 -20864.353} C_VEL
LIN {X 0,Y 213.889,Z 554.513,A -85,B 0,C 180,E1 -20866.702,E2 -20866.702} C_VEL
LIN {X 0,Y 212.925,Z 563.991,A -85,B 0,C 180,E1 -20869.54,E2 -20869.54} C_VEL
LIN {X 0,Y 212.272,Z 571.755,A -85,B 0,C 180,E1 -20872.389,E2 -20872.389} C_VEL
LIN {X 0,Y 211.875,Z 578.868,A -85,B 0,C 180,E1 -20875.634,E2 -20875.634} C_VEL
LIN {X 0,Y 211.836,Z 583.29,A -85,B 0,C 180,E1 -20878.098,E2 -20878.098} C_VEL
LIN {X 0,Y 211.85,Z 587.391,A -85,B 0,C 180,E1 -20880.95,E2 -20880.95} C_VEL
LIN {X 0,Y 212.253,Z 590.534,A -85,B 0,C 180,E1 -20883.797,E2 -20883.797} C_VEL
LIN {X 0,Y 213.079,Z 593.377,A -85,B 0,C 180,E1 -20887.581,E2 -20887.581} C_VEL
LIN {X 0,Y 214.933,Z 594.802,A -85,B 0,C 180,E1 -20891.314,E2 -20891.314} C_VEL
LIN {X 0,Y 217.518,Z 594.834,A -85,B 0,C 180,E1 -20894.98,E2 -20894.98} C_VEL
LIN {X 0,Y 221.284,Z 593.441,A -85,B 0,C 180,E1 -20898.518,E2 -20898.518} C_VEL
LIN {X 0,Y 225.766,Z 590.734,A -85,B 0,C 180,E1 -20901.935,E2 -20901.935} C_VEL
LIN {X 0,Y 231.236,Z 586.548,A -85,B 0,C 180,E1 -20905.182,E2 -20905.182} C_VEL
LIN {X 0,Y 237.596,Z 580.872,A -85,B 0,C 180,E1 -20908.247,E2 -20908.247} C_VEL
LIN {X 0,Y 244.768,Z 573.48,A -85,B 0,C 180,E1 -20911.12,E2 -20911.12} C_VEL
LIN {X 0,Y 250.634,Z 566.676,A -85,B 0,C 180,E1 -20913.147,E2 -20913.147} C_VEL
LIN {X 0,Y 251.344,Z 565.12,A -85,B 0,C 180,E1 -20914.003,E2 -20914.003} C_VEL
LIN {X 0,Y 252.254,Z 562.036,A -85,B 0,C 180,E1 -20916.102,E2 -20916.102} C_VEL
LIN {X 0,Y 252.679,Z 560.158,A -85,B 0,C 180,E1 -20917.727,E2 -20917.727} C_VEL
LIN {X 0,Y 252.77,Z 558.759,A -85,B 0,C 180,E1 -20919.754,E2 -20919.754} C_VEL
LIN {X 0,Y 252.876,Z 557.995,A -85,B 0,C 180,E1 -20921.837,E2 -20921.837} C_VEL
LIN {X 0,Y 252.98,Z 557.994,A -85,B 0,C 180,E1 -20923.989,E2 -20923.989} C_VEL
LIN {X 0,Y 252.883,Z 559.118,A -85,B 0,C 180,E1 -20926.268,E2 -20926.268} C_VEL
LIN {X 0,Y 252.66,Z 560.894,A -85,B 0,C 180,E1 -20928.119,E2 -20928.119} C_VEL
LIN {X 0,Y 252.258,Z 562.353,A -85,B 0,C 180,E1 -20929.079,E2 -20929.079} C_VEL
LIN {X 0,Y 251.097,Z 565.293,A -85,B 0,C 180,E1 -20930.502,E2 -20930.502} C_VEL
LIN {X 0,Y 247.284,Z 572.977,A -85,B 0,C 180,E1 -20933.356,E2 -20933.356} C_VEL
LIN {X 0,Y 242.176,Z 582.051,A -85,B 0,C 180,E1 -20936.538,E2 -20936.538} C_VEL
LIN {X 0,Y 237.528,Z 588.568,A -85,B 0,C 180,E1 -20938.816,E2 -20938.816} C_VEL
LIN {X 0,Y 230.709,Z 596.36,A -85,B 0,C 180,E1 -20941.825,E2 -20941.825} C_VEL
LIN {X 0,Y 229.34,Z 597.864,A -85,B 0,C 180,E1 -20942.513,E2 -20942.513} C_VEL
LIN {X 0,Y 227.204,Z 599.624,A -85,B 0,C 180,E1 -20943.242,E2 -20943.242} C_VEL
LIN {X 0,Y 217.532,Z 604.718,A -85,B 0,C 180,E1 -20945.294,E2 -20945.294} C_VEL
LIN {X 0,Y 215.588,Z 605.931,A -85,B 0,C 180,E1 -20946.147,E2 -20946.147} C_VEL
LIN {X 0,Y 212.483,Z 608.602,A -85,B 0,C 180,E1 -20948.664,E2 -20948.664} C_VEL
LIN {X 0,Y 208.866,Z 611.313,A -85,B 0,C 180,E1 -20952.372,E2 -20952.372} C_VEL
LIN {X 0,Y 206.33,Z 612.731,A -85,B 0,C 180,E1 -20956.206,E2 -20956.206} C_VEL
LIN {X 0,Y 205.116,Z 612.843,A -85,B 0,C 180,E1 -20960.136,E2 -20960.136} C_VEL
LIN {X 0,Y 204.877,Z 611.534,A -85,B 0,C 180,E1 -20964.153,E2 -20964.153} C_VEL
LIN {X 0,Y 205.351,Z 608.863,A -85,B 0,C 180,E1 -20968.039,E2 -20968.039} C_VEL
LIN {X 0,Y 205.704,Z 607.7,A -85,B 0,C 180,E1 -20969.388,E2 -20969.388} C_VEL
LIN {X 0,Y 205.258,Z 610.319,A -85,B 0,C 180,E1 -20971.962,E2 -20971.962} C_VEL
LIN {X 0,Y 204.824,Z 612.961,A -85,B 0,C 180,E1 -20975.908,E2 -20975.908} C_VEL
LIN {X 0,Y 205.115,Z 614.188,A -85,B 0,C 180,E1 -20979.865,E2 -20979.865} C_VEL
LIN {X 0,Y 206.34,Z 614.04,A -85,B 0,C 180,E1 -20983.793,E2 -20983.793} C_VEL
LIN {X 0,Y 208.853,Z 612.607,A -85,B 0,C 180,E1 -20987.629,E2 -20987.629} C_VEL
LIN {X 0,Y 212.412,Z 609.893,A -85,B 0,C 180,E1 -20991.343,E2 -20991.343} C_VEL
LIN {X 0,Y 217.292,Z 605.684,A -85,B 0,C 180,E1 -20995.094,E2 -20995.094} C_VEL
LIN {X 0,Y 222.862,Z 600.598,A -85,B 0,C 180,E1 -20998.231,E2 -20998.231} C_VEL
LIN {X 0,Y 229.783,Z 593.756,A -85,B 0,C 180,E1 -21001.329,E2 -21001.329} C_VEL
LIN {X 0,Y 235.284,Z 587.761,A -85,B 0,C 180,E1 -21003.546,E2 -21003.546} C_VEL
LIN {X 0,Y 238.055,Z 583.679,A -85,B 0,C 180,E1 -21005.148,E2 -21005.148} C_VEL
LIN {X 0,Y 241.297,Z 577.878,A -85,B 0,C 180,E1 -21007.709,E2 -21007.709} C_VEL
LIN {X 0,Y 243.152,Z 574.203,A -85,B 0,C 180,E1 -21009.486,E2 -21009.486} C_VEL
LIN {X 0,Y 244.83,Z 570.405,A -85,B 0,C 180,E1 -21011.725,E2 -21011.725} C_VEL
LIN {X 0,Y 245.454,Z 568.454,A -85,B 0,C 180,E1 -21013.408,E2 -21013.408} C_VEL
LIN {X 0,Y 246.054,Z 566.801,A -85,B 0,C 180,E1 -21015.567,E2 -21015.567} C_VEL
LIN {X 0,Y 246.189,Z 566.386,A -85,B 0,C 180,E1 -21016.754,E2 -21016.754} C_VEL
LIN {X 0,Y 246.021,Z 566.478,A -85,B 0,C 180,E1 -21018.926,E2 -21018.926} C_VEL
LIN {X 0,Y 245.956,Z 567.127,A -85,B 0,C 180,E1 -21021.051,E2 -21021.051} C_VEL
LIN {X 0,Y 245.79,Z 568.45,A -85,B 0,C 180,E1 -21023.189,E2 -21023.189} C_VEL
LIN {X 0,Y 245.353,Z 570.289,A -85,B 0,C 180,E1 -21025.048,E2 -21025.048} C_VEL
LIN {X 0,Y 244.902,Z 571.392,A -85,B 0,C 180,E1 -21025.972,E2 -21025.972} C_VEL
LIN {X 0,Y 243.479,Z 573.208,A -85,B 0,C 180,E1 -21026.741,E2 -21026.741} C_VEL
LIN {X 0,Y 237.525,Z 579.092,A -85,B 0,C 180,E1 -21028.816,E2 -21028.816} C_VEL
LIN {X 0,Y 230.163,Z 585.446,A -85,B 0,C 180,E1 -21031.752,E2 -21031.752} C_VEL
LIN {X 0,Y 223.774,Z 590.231,A -85,B 0,C 180,E1 -21034.914,E2 -21034.914} C_VEL
LIN {X 0,Y 219.56,Z 592.895,A -85,B 0,C 180,E1 -21037.412,E2 -21037.412} C_VEL
LIN {X 0,Y 214.797,Z 595.231,A -85,B 0,C 180,E1 -21040.902,E2 -21040.902} C_VEL
LIN {X 0,Y 210.986,Z 596.228,A -85,B 0,C 180,E1 -21044.545,E2 -21044.545} C_VEL
LIN {X 0,Y 208.047,Z 595.902,A -85,B 0,C 180,E1 -21048.306,E2 -21048.306} C_VEL
LIN {X 0,Y 206.159,Z 594.212,A -85,B 0,C 180,E1 -21052.163,E2 -21052.163} C_VEL
LIN {X 0,Y 205.246,Z 591.081,A -85,B 0,C 180,E1 -21056.074,E2 -21056.074} C_VEL
LIN {X 0,Y 204.765,Z 586.435,A -85,B 0,C 180,E1 -21060,E2 -21060} C_VEL
LIN {X 0,Y 204.817,Z 581.838,A -85,B 0,C 180,E1 -21062.951,E2 -21062.951} C_VEL
LIN {X 0,Y 204.983,Z 575.638,A -85,B 0,C 180,E1 -21066.126,E2 -21066.126} C_VEL
LIN {X 0,Y 205.554,Z 567.767,A -85,B 0,C 180,E1 -21069.347,E2 -21069.347} C_VEL
LIN {X 0,Y 206.428,Z 558.991,A -85,B 0,C 180,E1 -21072.286,E2 -21072.286} C_VEL
LIN {X 0,Y 207.352,Z 550.223,A -85,B 0,C 180,E1 -21074.727,E2 -21074.727} C_VEL
LIN {X 0,Y 208.607,Z 539.707,A -85,B 0,C 180,E1 -21077.145,E2 -21077.145} C_VEL
LIN {X 0,Y 209.843,Z 529.599,A -85,B 0,C 180,E1 -21079.06,E2 -21079.06} C_VEL
LIN {X 0,Y 210.713,Z 521.877,A -85,B 0,C 180,E1 -21080.314,E2 -21080.314} C_VEL
LIN {X 0,Y 208.407,Z 508.827,A -85,B 0,C 180,E1 -21082.145,E2 -21082.145} C_VEL
LIN {X 0,Y 206.247,Z 496.114,A -85,B 0,C 180,E1 -21083.589,E2 -21083.589} C_VEL
LIN {X 0,Y 205.419,Z 490.901,A -85,B 0,C 180,E1 -21084.114,E2 -21084.114} C_VEL
LIN {X 0,Y 205.784,Z 490.852,A -85,B 0,C 180,E1 -21088.564,E2 -21088.564} C_VEL
LIN {X 0,Y 206.272,Z 490.786,A -85,B 0,C 180,E1 -21093.035,E2 -21093.035} C_VEL
LIN {X 0,Y 206.475,Z 490.763,A -85,B 0,C 180,E1 -21095.356,E2 -21095.356} C_VEL
LIN {X 0,Y 206.63,Z 490.746,A -85,B 0,C 180,E1 -21098.529,E2 -21098.529} C_VEL
LIN {X 0,Y 206.624,Z 490.744,A -85,B 0,C 180,E1 -21102.866,E2 -21102.866} C_VEL
LIN {X 0,Y 206.63,Z 490.744,A -85,B 0,C 180,E1 -21107.136,E2 -21107.136} C_VEL
LIN {X 0,Y 206.705,Z 490.732,A -85,B 0,C 180,E1 -21111.446,E2 -21111.446} C_VEL
LIN {X 0,Y 206.735,Z 490.732,A -85,B 0,C 180,E1 -21114.695,E2 -21114.695} C_VEL
LIN {X 0,Y 206.727,Z 490.728,A -85,B 0,C 180,E1 -21119.34,E2 -21119.34} C_VEL
LIN {X 0,Y 206.737,Z 490.733,A -85,B 0,C 180,E1 -21123.773,E2 -21123.773} C_VEL
LIN {X 0,Y 206.762,Z 490.727,A -85,B 0,C 180,E1 -21128.044,E2 -21128.044} C_VEL
LIN {X 0,Y 206.878,Z 490.717,A -85,B 0,C 180,E1 -21132.197,E2 -21132.197} C_VEL
LIN {X 0,Y 206.919,Z 490.707,A -85,B 0,C 180,E1 -21136.246,E2 -21136.246} C_VEL
LIN {X 0,Y 207.137,Z 490.684,A -85,B 0,C 180,E1 -21140.233,E2 -21140.233} C_VEL
LIN {X 0,Y 207.194,Z 490.676,A -85,B 0,C 180,E1 -21142.202,E2 -21142.202} C_VEL
LIN {X 0,Y 207.387,Z 490.652,A -85,B 0,C 180,E1 -21148.058,E2 -21148.058} C_VEL
LIN {X 0,Y 207.52,Z 490.637,A -85,B 0,C 180,E1 -21150,E2 -21150} C_VEL
LIN {X 0,Y 207.385,Z 490.653,A -85,B 0,C 180,E1 -21151.942,E2 -21151.942} C_VEL
LIN {X 0,Y 207.137,Z 490.683,A -85,B 0,C 180,E1 -21157.8,E2 -21157.8} C_VEL
LIN {X 0,Y 206.936,Z 490.708,A -85,B 0,C 180,E1 -21161.758,E2 -21161.758} C_VEL
LIN {X 0,Y 206.872,Z 490.716,A -85,B 0,C 180,E1 -21165.77,E2 -21165.77} C_VEL
LIN {X 0,Y 206.788,Z 490.726,A -85,B 0,C 180,E1 -21169.869,E2 -21169.869} C_VEL
LIN {X 0,Y 206.767,Z 490.729,A -85,B 0,C 180,E1 -21174.072,E2 -21174.072} C_VEL
LIN {X 0,Y 206.748,Z 490.729,A -85,B 0,C 180,E1 -21178.418,E2 -21178.418} C_VEL
LIN {X 0,Y 206.713,Z 490.733,A -85,B 0,C 180,E1 -21182.955,E2 -21182.955} C_VEL
LIN {X 0,Y 206.725,Z 490.734,A -85,B 0,C 180,E1 -21185.32,E2 -21185.32} C_VEL
LIN {X 0,Y 206.67,Z 490.738,A -85,B 0,C 180,E1 -21190.249,E2 -21190.249} C_VEL
LIN {X 0,Y 206.637,Z 490.746,A -85,B 0,C 180,E1 -21195.581,E2 -21195.581} C_VEL
LIN {X 0,Y 206.656,Z 490.742,A -85,B 0,C 180,E1 -21199.747,E2 -21199.747} C_VEL
LIN {X 0,Y 206.657,Z 490.742,A -85,B 0,C 180,E1 -21202.254,E2 -21202.254} C_VEL
LIN {X 0,Y 206.532,Z 490.756,A -85,B 0,C 180,E1 -21204.755,E2 -21204.755} C_VEL
LIN {X 0,Y 206.174,Z 490.801,A -85,B 0,C 180,E1 -21209.248,E2 -21209.248} C_VEL
LIN {X 0,Y 205.632,Z 490.87,A -85,B 0,C 180,E1 -21213.62,E2 -21213.62} C_VEL
LIN {X 0,Y 205.406,Z 490.914,A -85,B 0,C 180,E1 -21216.255,E2 -21216.255} C_VEL
LIN {X 0,Y 207.674,Z 504.531,A -85,B 0,C 180,E1 -21217.665,E2 -21217.665} C_VEL
LIN {X 0,Y 210.076,Z 518.497,A -85,B 0,C 180,E1 -21219.51,E2 -21219.51} C_VEL
LIN {X 0,Y 210.56,Z 521.075,A -85,B 0,C 180,E1 -21219.906,E2 -21219.906} C_VEL
LIN {X 0,Y 209.304,Z 533.1,A -85,B 0,C 180,E1 -21221.904,E2 -21221.904} C_VEL
LIN {X 0,Y 207.877,Z 544.679,A -85,B 0,C 180,E1 -21224.307,E2 -21224.307} C_VEL
LIN {X 0,Y 206.783,Z 554.281,A -85,B 0,C 180,E1 -21226.737,E2 -21226.737} C_VEL
LIN {X 0,Y 205.815,Z 563.808,A -85,B 0,C 180,E1 -21229.672,E2 -21229.672} C_VEL
LIN {X 0,Y 205.169,Z 571.678,A -85,B 0,C 180,E1 -21232.619,E2 -21232.619} C_VEL
LIN {X 0,Y 204.803,Z 579.094,A -85,B 0,C 180,E1 -21236.064,E2 -21236.064} C_VEL
LIN {X 0,Y 204.727,Z 584.109,A -85,B 0,C 180,E1 -21239.016,E2 -21239.016} C_VEL
LIN {X 0,Y 205.026,Z 589.256,A -85,B 0,C 180,E1 -21242.947,E2 -21242.947} C_VEL
LIN {X 0,Y 205.536,Z 592.042,A -85,B 0,C 180,E1 -21245.887,E2 -21245.887} C_VEL
LIN {X 0,Y 206.887,Z 594.502,A -85,B 0,C 180,E1 -21249.779,E2 -21249.779} C_VEL
LIN {X 0,Y 209.315,Z 595.522,A -85,B 0,C 180,E1 -21253.593,E2 -21253.593} C_VEL
LIN {X 0,Y 212.524,Z 595.21,A -85,B 0,C 180,E1 -21257.314,E2 -21257.314} C_VEL
LIN {X 0,Y 216.819,Z 593.557,A -85,B 0,C 180,E1 -21260.888,E2 -21260.888} C_VEL
LIN {X 0,Y 222.115,Z 590.48,A -85,B 0,C 180,E1 -21264.288,E2 -21264.288} C_VEL
LIN {X 0,Y 228.237,Z 586.063,A -85,B 0,C 180,E1 -21267.509,E2 -21267.509} C_VEL
LIN {X 0,Y 235.281,Z 580.064,A -85,B 0,C 180,E1 -21270.517,E2 -21270.517} C_VEL
LIN {X 0,Y 243.138,Z 572.396,A -85,B 0,C 180,E1 -21273.312,E2 -21273.312} C_VEL
LIN {X 0,Y 245.155,Z 570.221,A -85,B 0,C 180,E1 -21273.988,E2 -21273.988} C_VEL
LIN {X 0,Y 246.082,Z 568.657,A -85,B 0,C 180,E1 -21274.833,E2 -21274.833} C_VEL
LIN {X 0,Y 247.247,Z 565.676,A -85,B 0,C 180,E1 -21277.259,E2 -21277.259} C_VEL
LIN {X 0,Y 247.634,Z 564.506,A -85,B 0,C 180,E1 -21278.636,E2 -21278.636} C_VEL
LIN {X 0,Y 247.834,Z 563.466,A -85,B 0,C 180,E1 -21280.709,E2 -21280.709} C_VEL
LIN {X 0,Y 247.994,Z 563.106,A -85,B 0,C 180,E1 -21282.855,E2 -21282.855} C_VEL
LIN {X 0,Y 247.994,Z 563.688,A -85,B 0,C 180,E1 -21285.112,E2 -21285.112} C_VEL
LIN {X 0,Y 247.696,Z 565.503,A -85,B 0,C 180,E1 -21287.537,E2 -21287.537} C_VEL
LIN {X 0,Y 247.223,Z 566.833,A -85,B 0,C 180,E1 -21288.554,E2 -21288.554} C_VEL
LIN {X 0,Y 245.813,Z 569.682,A -85,B 0,C 180,E1 -21289.962,E2 -21289.962} C_VEL
LIN {X 0,Y 241.466,Z 576.981,A -85,B 0,C 180,E1 -21292.847,E2 -21292.847} C_VEL
LIN {X 0,Y 236.611,Z 584.317,A -85,B 0,C 180,E1 -21295.642,E2 -21295.642} C_VEL
LIN {X 0,Y 231.644,Z 590.437,A -85,B 0,C 180,E1 -21297.931,E2 -21297.931} C_VEL
LIN {X 0,Y 224.578,Z 597.682,A -85,B 0,C 180,E1 -21300.983,E2 -21300.983} C_VEL
LIN {X 0,Y 219.308,Z 602.687,A -85,B 0,C 180,E1 -21303.805,E2 -21303.805} C_VEL
LIN {X 0,Y 215.588,Z 605.931,A -85,B 0,C 180,E1 -21306.147,E2 -21306.147} C_VEL
LIN {X 0,Y 213.117,Z 607.603,A -85,B 0,C 180,E1 -21307.517,E2 -21307.517} C_VEL
LIN {X 0,Y 207.679,Z 609.816,A -85,B 0,C 180,E1 -21309.698,E2 -21309.698} C_VEL
LIN {X 0,Y 202.578,Z 611.298,A -85,B 0,C 180,E1 -21312.028,E2 -21312.028} C_VEL
LIN {X 0,Y 200.684,Z 611.836,A -85,B 0,C 180,E1 -21313.603,E2 -21313.603} C_VEL
LIN {X 0,Y 199.419,Z 612.249,A -85,B 0,C 180,E1 -21315.718,E2 -21315.718} C_VEL
LIN {X 0,Y 198.135,Z 612.042,A -85,B 0,C 180,E1 -21319.784,E2 -21319.784} C_VEL
LIN {X 0,Y 197.867,Z 610.476,A -85,B 0,C 180,E1 -21324,E2 -21324} C_VEL
LIN {X 0,Y 198.366,Z 607.547,A -85,B 0,C 180,E1 -21327.97,E2 -21327.97} C_VEL
LIN {X 0,Y 198.738,Z 606.265,A -85,B 0,C 180,E1 -21329.43,E2 -21329.43} C_VEL
LIN {X 0,Y 198.272,Z 609.009,A -85,B 0,C 180,E1 -21332.031,E2 -21332.031} C_VEL
LIN {X 0,Y 197.805,Z 611.922,A -85,B 0,C 180,E1 -21336.119,E2 -21336.119} C_VEL
LIN {X 0,Y 198.135,Z 613.38,A -85,B 0,C 180,E1 -21340.216,E2 -21340.216} C_VEL
LIN {X 0,Y 199.429,Z 613.546,A -85,B 0,C 180,E1 -21344.281,E2 -21344.281} C_VEL
LIN {X 0,Y 202.099,Z 612.46,A -85,B 0,C 180,E1 -21348.239,E2 -21348.239} C_VEL
LIN {X 0,Y 205.821,Z 610.13,A -85,B 0,C 180,E1 -21352.062,E2 -21352.062} C_VEL
LIN {X 0,Y 210.605,Z 606.527,A -85,B 0,C 180,E1 -21355.71,E2 -21355.71} C_VEL
LIN {X 0,Y 216.709,Z 601.635,A -85,B 0,C 180,E1 -21359.108,E2 -21359.108} C_VEL
LIN {X 0,Y 223.877,Z 595.37,A -85,B 0,C 180,E1 -21362.254,E2 -21362.254} C_VEL
LIN {X 0,Y 229.624,Z 589.722,A -85,B 0,C 180,E1 -21364.487,E2 -21364.487} C_VEL
LIN {X 0,Y 232.589,Z 586.017,A -85,B 0,C 180,E1 -21366.102,E2 -21366.102} C_VEL
LIN {X 0,Y 236.08,Z 580.652,A -85,B 0,C 180,E1 -21368.694,E2 -21368.694} C_VEL
LIN {X 0,Y 238.716,Z 576.177,A -85,B 0,C 180,E1 -21371.144,E2 -21371.144} C_VEL
LIN {X 0,Y 239.775,Z 573.899,A -85,B 0,C 180,E1 -21372.881,E2 -21372.881} C_VEL
LIN {X 0,Y 240.463,Z 572.355,A -85,B 0,C 180,E1 -21374.543,E2 -21374.543} C_VEL
LIN {X 0,Y 240.956,Z 571.16,A -85,B 0,C 180,E1 -21376.818,E2 -21376.818} C_VEL
LIN {X 0,Y 240.661,Z 571.481,A -85,B 0,C 180,E1 -21380.024,E2 -21380.024} C_VEL
LIN {X 0,Y 240.395,Z 572.397,A -85,B 0,C 180,E1 -21382.125,E2 -21382.125} C_VEL
LIN {X 0,Y 239.888,Z 573.868,A -85,B 0,C 180,E1 -21384.131,E2 -21384.131} C_VEL
LIN {X 0,Y 239.4,Z 575.005,A -85,B 0,C 180,E1 -21385.285,E2 -21385.285} C_VEL
LIN {X 0,Y 235.859,Z 578.318,A -85,B 0,C 180,E1 -21386.546,E2 -21386.546} C_VEL
LIN {X 0,Y 227.904,Z 584.961,A -85,B 0,C 180,E1 -21389.415,E2 -21389.415} C_VEL
LIN {X 0,Y 220.766,Z 589.983,A -85,B 0,C 180,E1 -21392.51,E2 -21392.51} C_VEL
LIN {X 0,Y 216.059,Z 592.834,A -85,B 0,C 180,E1 -21394.985,E2 -21394.985} C_VEL
LIN {X 0,Y 210.532,Z 595.445,A -85,B 0,C 180,E1 -21398.457,E2 -21398.457} C_VEL
LIN {X 0,Y 206.012,Z 596.75,A -85,B 0,C 180,E1 -21402.12,E2 -21402.12} C_VEL
LIN {X 0,Y 202.595,Z 596.744,A -85,B 0,C 180,E1 -21405.947,E2 -21405.947} C_VEL
LIN {X 0,Y 199.965,Z 595.382,A -85,B 0,C 180,E1 -21409.879,E2 -21409.879} C_VEL
LIN {X 0,Y 198.593,Z 592.658,A -85,B 0,C 180,E1 -21413.906,E2 -21413.906} C_VEL
LIN {X 0,Y 197.995,Z 589.678,A -85,B 0,C 180,E1 -21416.948,E2 -21416.948} C_VEL
LIN {X 0,Y 197.699,Z 585.803,A -85,B 0,C 180,E1 -21420,E2 -21420} C_VEL
LIN {X 0,Y 197.755,Z 580.93,A -85,B 0,C 180,E1 -21423.056,E2 -21423.056} C_VEL
LIN {X 0,Y 197.949,Z 574.705,A -85,B 0,C 180,E1 -21426.218,E2 -21426.218} C_VEL
LIN {X 0,Y 198.47,Z 567.645,A -85,B 0,C 180,E1 -21429.17,E2 -21429.17} C_VEL
LIN {X 0,Y 199.309,Z 558.751,A -85,B 0,C 180,E1 -21432.215,E2 -21432.215} C_VEL
LIN {X 0,Y 200.517,Z 547.849,A -85,B 0,C 180,E1 -21435.241,E2 -21435.241} C_VEL
LIN {X 0,Y 201.829,Z 536.853,A -85,B 0,C 180,E1 -21437.74,E2 -21437.74} C_VEL
LIN {X 0,Y 202.928,Z 527.688,A -85,B 0,C 180,E1 -21439.472,E2 -21439.472} C_VEL
LIN {X 0,Y 203.496,Z 521.554,A -85,B 0,C 180,E1 -21440.481,E2 -21440.481} C_VEL
LIN {X 0,Y 200.948,Z 507.327,A -85,B 0,C 180,E1 -21442.509,E2 -21442.509} C_VEL
LIN {X 0,Y 198.637,Z 493.116,A -85,B 0,C 180,E1 -21444.085,E2 -21444.085} C_VEL
LIN {X 0,Y 198.397,Z 491.775,A -85,B 0,C 180,E1 -21444.257,E2 -21444.257} C_VEL
LIN {X 0,Y 198.683,Z 491.739,A -85,B 0,C 180,E1 -21447.831,E2 -21447.831} C_VEL
LIN {X 0,Y 199.139,Z 491.678,A -85,B 0,C 180,E1 -21452.112,E2 -21452.112} C_VEL
LIN {X 0,Y 199.445,Z 491.64,A -85,B 0,C 180,E1 -21455.858,E2 -21455.858} C_VEL
LIN {X 0,Y 199.583,Z 491.621,A -85,B 0,C 180,E1 -21459.335,E2 -21459.335} C_VEL
LIN {X 0,Y 199.573,Z 491.622,A -85,B 0,C 180,E1 -21462.309,E2 -21462.309} C_VEL
LIN {X 0,Y 199.583,Z 491.622,A -85,B 0,C 180,E1 -21465.229,E2 -21465.229} C_VEL
LIN {X 0,Y 199.642,Z 491.613,A -85,B 0,C 180,E1 -21470.68,E2 -21470.68} C_VEL
LIN {X 0,Y 199.639,Z 491.616,A -85,B 0,C 180,E1 -21475.718,E2 -21475.718} C_VEL
LIN {X 0,Y 199.708,Z 491.606,A -85,B 0,C 180,E1 -21478.138,E2 -21478.138} C_VEL
LIN {X 0,Y 199.691,Z 491.609,A -85,B 0,C 180,E1 -21482.772,E2 -21482.772} C_VEL
LIN {X 0,Y 199.742,Z 491.6,A -85,B 0,C 180,E1 -21487.23,E2 -21487.23} C_VEL
LIN {X 0,Y 199.801,Z 491.596,A -85,B 0,C 180,E1 -21491.757,E2 -21491.757} C_VEL
LIN {X 0,Y 199.853,Z 491.589,A -85,B 0,C 180,E1 -21495.749,E2 -21495.749} C_VEL
LIN {X 0,Y 200.08,Z 491.562,A -85,B 0,C 180,E1 -21499.885,E2 -21499.885} C_VEL
LIN {X 0,Y 200.137,Z 491.556,A -85,B 0,C 180,E1 -21501.925,E2 -21501.925} C_VEL
LIN {X 0,Y 200.327,Z 491.531,A -85,B 0,C 180,E1 -21507.989,E2 -21507.989} C_VEL
LIN {X 0,Y 200.484,Z 491.514,A -85,B 0,C 180,E1 -21510,E2 -21510} C_VEL
LIN {X 0,Y 200.026,Z 491.566,A -85,B 0,C 180,E1 -21514.03,E2 -21514.03} C_VEL
LIN {X 0,Y 200.086,Z 491.563,A -85,B 0,C 180,E1 -21518.077,E2 -21518.077} C_VEL
LIN {X 0,Y 199.884,Z 491.583,A -85,B 0,C 180,E1 -21522.179,E2 -21522.179} C_VEL
LIN {X 0,Y 199.809,Z 491.595,A -85,B 0,C 180,E1 -21526.343,E2 -21526.343} C_VEL
LIN {X 0,Y 199.704,Z 491.605,A -85,B 0,C 180,E1 -21530.605,E2 -21530.605} C_VEL
LIN {X 0,Y 199.677,Z 491.61,A -85,B 0,C 180,E1 -21534.984,E2 -21534.984} C_VEL
LIN {X 0,Y 199.678,Z 491.611,A -85,B 0,C 180,E1 -21539.522,E2 -21539.522} C_VEL
LIN {X 0,Y 199.668,Z 491.611,A -85,B 0,C 180,E1 -21542.352,E2 -21542.352} C_VEL
LIN {X 0,Y 199.643,Z 491.614,A -85,B 0,C 180,E1 -21546.759,E2 -21546.759} C_VEL
LIN {X 0,Y 199.642,Z 491.613,A -85,B 0,C 180,E1 -21549.32,E2 -21549.32} C_VEL
LIN {X 0,Y 199.583,Z 491.622,A -85,B 0,C 180,E1 -21554.771,E2 -21554.771} C_VEL
LIN {X 0,Y 199.58,Z 491.621,A -85,B 0,C 180,E1 -21558.004,E2 -21558.004} C_VEL
LIN {X 0,Y 199.599,Z 491.619,A -85,B 0,C 180,E1 -21560.772,E2 -21560.772} C_VEL
LIN {X 0,Y 199.497,Z 491.633,A -85,B 0,C 180,E1 -21564.122,E2 -21564.122} C_VEL
LIN {X 0,Y 199.226,Z 491.666,A -85,B 0,C 180,E1 -21568.051,E2 -21568.051} C_VEL
LIN {X 0,Y 198.718,Z 491.73,A -85,B 0,C 180,E1 -21572.627,E2 -21572.627} C_VEL
LIN {X 0,Y 198.388,Z 491.771,A -85,B 0,C 180,E1 -21576.138,E2 -21576.138} C_VEL
LIN {X 0,Y 200.583,Z 505.243,A -85,B 0,C 180,E1 -21577.592,E2 -21577.592} C_VEL
LIN {X 0,Y 202.813,Z 518.028,A -85,B 0,C 180,E1 -21579.329,E2 -21579.329} C_VEL
LIN {X 0,Y 203.352,Z 522.615,A -85,B 0,C 180,E1 -21580.044,E2 -21580.044} C_VEL
LIN {X 0,Y 202.042,Z 533.789,A -85,B 0,C 180,E1 -21582.018,E2 -21582.018} C_VEL
LIN {X 0,Y 200.668,Z 545.253,A -85,B 0,C 180,E1 -21584.511,E2 -21584.511} C_VEL
LIN {X 0,Y 199.538,Z 555.703,A -85,B 0,C 180,E1 -21587.283,E2 -21587.283} C_VEL
LIN {X 0,Y 198.572,Z 565.06,A -85,B 0,C 180,E1 -21590.321,E2 -21590.321} C_VEL
LIN {X 0,Y 197.98,Z 572.743,A -85,B 0,C 180,E1 -21593.374,E2 -21593.374} C_VEL
LIN {X 0,Y 197.749,Z 579.944,A -85,B 0,C 180,E1 -21596.944,E2 -21596.944} C_VEL
LIN {X 0,Y 197.676,Z 584.891,A -85,B 0,C 180,E1 -21600,E2 -21600} C_VEL
LIN {X 0,Y 197.969,Z 588.833,A -85,B 0,C 180,E1 -21603.052,E2 -21603.052} C_VEL
LIN {X 0,Y 198.472,Z 591.86,A -85,B 0,C 180,E1 -21606.098,E2 -21606.098} C_VEL
LIN {X 0,Y 199.897,Z 594.616,A -85,B 0,C 180,E1 -21610.124,E2 -21610.124} C_VEL
LIN {X 0,Y 202.435,Z 596.006,A -85,B 0,C 180,E1 -21614.064,E2 -21614.064} C_VEL
LIN {X 0,Y 203.914,Z 596.206,A -85,B 0,C 180,E1 -21616.005,E2 -21616.005} C_VEL
LIN {X 0,Y 208.046,Z 595.535,A -85,B 0,C 180,E1 -21619.743,E2 -21619.743} C_VEL
LIN {X 0,Y 212.946,Z 593.587,A -85,B 0,C 180,E1 -21623.331,E2 -21623.331} C_VEL
LIN {X 0,Y 218.91,Z 590.3,A -85,B 0,C 180,E1 -21626.709,E2 -21626.709} C_VEL
LIN {X 0,Y 225.755,Z 585.581,A -85,B 0,C 180,E1 -21629.874,E2 -21629.874} C_VEL
LIN {X 0,Y 233.494,Z 579.36,A -85,B 0,C 180,E1 -21632.805,E2 -21632.805} C_VEL
LIN {X 0,Y 239.767,Z 573.57,A -85,B 0,C 180,E1 -21634.86,E2 -21634.86} C_VEL
LIN {X 0,Y 240.824,Z 572.159,A -85,B 0,C 180,E1 -21635.708,E2 -21635.708} C_VEL
LIN {X 0,Y 241.893,Z 570.115,A -85,B 0,C 180,E1 -21637.599,E2 -21637.599} C_VEL
LIN {X 0,Y 242.45,Z 568.755,A -85,B 0,C 180,E1 -21639.622,E2 -21639.622} C_VEL
LIN {X 0,Y 242.723,Z 568.113,A -85,B 0,C 180,E1 -21641.756,E2 -21641.756} C_VEL
LIN {X 0,Y 242.828,Z 568.25,A -85,B 0,C 180,E1 -21643.996,E2 -21643.996} C_VEL
LIN {X 0,Y 242.602,Z 569.497,A -85,B 0,C 180,E1 -21646.405,E2 -21646.405} C_VEL
LIN {X 0,Y 242.012,Z 571.282,A -85,B 0,C 180,E1 -21648.093,E2 -21648.093} C_VEL
LIN {X 0,Y 239.701,Z 574.834,A -85,B 0,C 180,E1 -21649.831,E2 -21649.831} C_VEL
LIN {X 0,Y 235.546,Z 580.705,A -85,B 0,C 180,E1 -21652.29,E2 -21652.29} C_VEL
LIN {X 0,Y 231.071,Z 586.518,A -85,B 0,C 180,E1 -21654.698,E2 -21654.698} C_VEL
LIN {X 0,Y 227.688,Z 590.342,A -85,B 0,C 180,E1 -21656.248,E2 -21656.248} C_VEL
LIN {X 0,Y 220.234,Z 597.361,A -85,B 0,C 180,E1 -21659.297,E2 -21659.297} C_VEL
LIN {X 0,Y 213.709,Z 602.944,A -85,B 0,C 180,E1 -21662.587,E2 -21662.587} C_VEL
LIN {X 0,Y 209.046,Z 606.499,A -85,B 0,C 180,E1 -21665.442,E2 -21665.442} C_VEL
LIN {X 0,Y 205.891,Z 608.862,A -85,B 0,C 180,E1 -21667.946,E2 -21667.946} C_VEL
LIN {X 0,Y 202.115,Z 611.189,A -85,B 0,C 180,E1 -21671.763,E2 -21671.763} C_VEL
LIN {X 0,Y 200.684,Z 611.836,A -85,B 0,C 180,E1 -21673.603,E2 -21673.603} C_VEL
LIN {X 0,Y 198.998,Z 612.196,A -85,B 0,C 180,E1 -21675.225,E2 -21675.225} C_VEL
LIN {X 0,Y 195.024,Z 611.951,A -85,B 0,C 180,E1 -21677.868,E2 -21677.868} C_VEL
LIN {X 0,Y 192.138,Z 611.157,A -85,B 0,C 180,E1 -21680.047,E2 -21680.047} C_VEL
LIN {X 0,Y 190.947,Z 610.352,A -85,B 0,C 180,E1 -21681.764,E2 -21681.764} C_VEL
LIN {X 0,Y 190.847,Z 610.031,A -85,B 0,C 180,E1 -21682.349,E2 -21682.349} C_VEL
LIN {X 0,Y 191.006,Z 607.944,A -85,B 0,C 180,E1 -21685.78,E2 -21685.78} C_VEL
LIN {X 0,Y 191.831,Z 604.683,A -85,B 0,C 180,E1 -21689.41,E2 -21689.41} C_VEL
LIN {X 0,Y 191.31,Z 607.597,A -85,B 0,C 180,E1 -21692.105,E2 -21692.105} C_VEL
LIN {X 0,Y 190.811,Z 610.755,A -85,B 0,C 180,E1 -21696.344,E2 -21696.344} C_VEL
LIN {X 0,Y 191.17,Z 612.541,A -85,B 0,C 180,E1 -21700.592,E2 -21700.592} C_VEL
LIN {X 0,Y 192.54,Z 612.999,A -85,B 0,C 180,E1 -21704.804,E2 -21704.804} C_VEL
LIN {X 0,Y 195.354,Z 612.228,A -85,B 0,C 180,E1 -21708.892,E2 -21708.892} C_VEL
LIN {X 0,Y 199.267,Z 610.232,A -85,B 0,C 180,E1 -21712.828,E2 -21712.828} C_VEL
LIN {X 0,Y 204.262,Z 607.052,A -85,B 0,C 180,E1 -21716.57,E2 -21716.57} C_VEL
LIN {X 0,Y 210.605,Z 602.609,A -85,B 0,C 180,E1 -21720.037,E2 -21720.037} C_VEL
LIN {X 0,Y 218.019,Z 596.856,A -85,B 0,C 180,E1 -21723.231,E2 -21723.231} C_VEL
LIN {X 0,Y 224.002,Z 591.676,A -85,B 0,C 180,E1 -21725.481,E2 -21725.481} C_VEL
LIN {X 0,Y 225.717,Z 589.91,A -85,B 0,C 180,E1 -21726.27,E2 -21726.27} C_VEL
LIN {X 0,Y 229.697,Z 584.886,A -85,B 0,C 180,E1 -21728.847,E2 -21728.847} C_VEL
LIN {X 0,Y 233.021,Z 580.217,A -85,B 0,C 180,E1 -21731.57,E2 -21731.57} C_VEL
LIN {X 0,Y 233.89,Z 578.881,A -85,B 0,C 180,E1 -21732.539,E2 -21732.539} C_VEL
LIN {X 0,Y 234.612,Z 577.421,A -85,B 0,C 180,E1 -21734.033,E2 -21734.033} C_VEL
LIN {X 0,Y 235.295,Z 576.1,A -85,B 0,C 180,E1 -21735.796,E2 -21735.796} C_VEL
LIN {X 0,Y 235.434,Z 575.797,A -85,B 0,C 180,E1 -21736.64,E2 -21736.64} C_VEL
LIN {X 0,Y 235.221,Z 575.746,A -85,B 0,C 180,E1 -21738.904,E2 -21738.904} C_VEL
LIN {X 0,Y 234.864,Z 576.315,A -85,B 0,C 180,E1 -21741.08,E2 -21741.08} C_VEL
LIN {X 0,Y 233.95,Z 578.174,A -85,B 0,C 180,E1 -21744.204,E2 -21744.204} C_VEL
LIN {X 0,Y 232.515,Z 579.548,A -85,B 0,C 180,E1 -21744.95,E2 -21744.95} C_VEL
LIN {X 0,Y 224.094,Z 585.948,A -85,B 0,C 180,E1 -21747.782,E2 -21747.782} C_VEL
LIN {X 0,Y 216.443,Z 590.887,A -85,B 0,C 180,E1 -21750.853,E2 -21750.853} C_VEL
LIN {X 0,Y 209.799,Z 594.403,A -85,B 0,C 180,E1 -21754.184,E2 -21754.184} C_VEL
LIN {X 0,Y 204.042,Z 596.598,A -85,B 0,C 180,E1 -21757.736,E2 -21757.736} C_VEL
LIN {X 0,Y 199.322,Z 597.509,A -85,B 0,C 180,E1 -21761.499,E2 -21761.499} C_VEL
LIN {X 0,Y 195.725,Z 597.131,A -85,B 0,C 180,E1 -21765.443,E2 -21765.443} C_VEL
LIN {X 0,Y 192.983,Z 595.46,A -85,B 0,C 180,E1 -21769.509,E2 -21769.509} C_VEL
LIN {X 0,Y 191.548,Z 592.414,A -85,B 0,C 180,E1 -21773.681,E2 -21773.681} C_VEL
LIN {X 0,Y 190.939,Z 589.194,A -85,B 0,C 180,E1 -21776.836,E2 -21776.836} C_VEL
LIN {X 0,Y 190.621,Z 583.474,A -85,B 0,C 180,E1 -21781.057,E2 -21781.057} C_VEL
LIN {X 0,Y 190.719,Z 577.961,A -85,B 0,C 180,E1 -21784.227,E2 -21784.227} C_VEL
LIN {X 0,Y 191.202,Z 570.012,A -85,B 0,C 180,E1 -21787.923,E2 -21787.923} C_VEL
LIN {X 0,Y 191.907,Z 561.583,A -85,B 0,C 180,E1 -21791.086,E2 -21791.086} C_VEL
LIN {X 0,Y 192.773,Z 553.223,A -85,B 0,C 180,E1 -21793.709,E2 -21793.709} C_VEL
LIN {X 0,Y 194.148,Z 542.155,A -85,B 0,C 180,E1 -21796.564,E2 -21796.564} C_VEL
LIN {X 0,Y 195.645,Z 529.747,A -85,B 0,C 180,E1 -21799.135,E2 -21799.135} C_VEL
LIN {X 0,Y 196.385,Z 522.393,A -85,B 0,C 180,E1 -21800.422,E2 -21800.422} C_VEL
LIN {X 0,Y 193.943,Z 508.416,A -85,B 0,C 180,E1 -21802.505,E2 -21802.505} C_VEL
LIN {X 0,Y 191.663,Z 494.278,A -85,B 0,C 180,E1 -21804.159,E2 -21804.159} C_VEL
LIN {X 0,Y 191.347,Z 492.652,A -85,B 0,C 180,E1 -21804.349,E2 -21804.349} C_VEL
LIN {X 0,Y 191.672,Z 492.611,A -85,B 0,C 180,E1 -21808.469,E2 -21808.469} C_VEL
LIN {X 0,Y 192.154,Z 492.544,A -85,B 0,C 180,E1 -21813.273,E2 -21813.273} C_VEL
LIN {X 0,Y 192.414,Z 492.518,A -85,B 0,C 180,E1 -21816.528,E2 -21816.528} C_VEL
LIN {X 0,Y 192.506,Z 492.5,A -85,B 0,C 180,E1 -21821.083,E2 -21821.083} C_VEL
LIN {X 0,Y 192.516,Z 492.505,A -85,B 0,C 180,E1 -21826.083,E2 -21826.083} C_VEL
LIN {X 0,Y 192.544,Z 492.498,A -85,B 0,C 180,E1 -21830.043,E2 -21830.043} C_VEL
LIN {X 0,Y 192.602,Z 492.495,A -85,B 0,C 180,E1 -21834.279,E2 -21834.279} C_VEL
LIN {X 0,Y 192.611,Z 492.486,A -85,B 0,C 180,E1 -21839.281,E2 -21839.281} C_VEL
LIN {X 0,Y 192.668,Z 492.483,A -85,B 0,C 180,E1 -21841.692,E2 -21841.692} C_VEL
LIN {X 0,Y 192.71,Z 492.478,A -85,B 0,C 180,E1 -21846.349,E2 -21846.349} C_VEL
LIN {X 0,Y 192.736,Z 492.475,A -85,B 0,C 180,E1 -21851.457,E2 -21851.457} C_VEL
LIN {X 0,Y 192.777,Z 492.469,A -85,B 0,C 180,E1 -21855.215,E2 -21855.215} C_VEL
LIN {X 0,Y 193.024,Z 492.439,A -85,B 0,C 180,E1 -21859.511,E2 -21859.511} C_VEL
LIN {X 0,Y 193.009,Z 492.442,A -85,B 0,C 180,E1 -21863.729,E2 -21863.729} C_VEL
LIN {X 0,Y 193.269,Z 492.41,A -85,B 0,C 180,E1 -21867.916,E2 -21867.916} C_VEL
LIN {X 0,Y 193.448,Z 492.39,A -85,B 0,C 180,E1 -21870,E2 -21870} C_VEL
LIN {X 0,Y 192.972,Z 492.444,A -85,B 0,C 180,E1 -21874.177,E2 -21874.177} C_VEL
LIN {X 0,Y 193.035,Z 492.439,A -85,B 0,C 180,E1 -21878.374,E2 -21878.374} C_VEL
LIN {X 0,Y 192.809,Z 492.462,A -85,B 0,C 180,E1 -21882.633,E2 -21882.633} C_VEL
LIN {X 0,Y 192.762,Z 492.472,A -85,B 0,C 180,E1 -21886.958,E2 -21886.958} C_VEL
LIN {X 0,Y 192.641,Z 492.485,A -85,B 0,C 180,E1 -21891.397,E2 -21891.397} C_VEL
LIN {X 0,Y 192.668,Z 492.485,A -85,B 0,C 180,E1 -21894.224,E2 -21894.224} C_VEL
LIN {X 0,Y 192.654,Z 492.484,A -85,B 0,C 180,E1 -21898.892,E2 -21898.892} C_VEL
LIN {X 0,Y 192.604,Z 492.491,A -85,B 0,C 180,E1 -21903.185,E2 -21903.185} C_VEL
LIN {X 0,Y 192.613,Z 492.49,A -85,B 0,C 180,E1 -21906.607,E2 -21906.607} C_VEL
LIN {X 0,Y 192.527,Z 492.499,A -85,B 0,C 180,E1 -21911.077,E2 -21911.077} C_VEL
LIN {X 0,Y 192.494,Z 492.505,A -85,B 0,C 180,E1 -21916.076,E2 -21916.076} C_VEL
LIN {X 0,Y 192.511,Z 492.504,A -85,B 0,C 180,E1 -21920.054,E2 -21920.054} C_VEL
LIN {X 0,Y 192.434,Z 492.513,A -85,B 0,C 180,E1 -21924.242,E2 -21924.242} C_VEL
LIN {X 0,Y 192.017,Z 492.564,A -85,B 0,C 180,E1 -21929.175,E2 -21929.175} C_VEL
LIN {X 0,Y 191.51,Z 492.628,A -85,B 0,C 180,E1 -21933.872,E2 -21933.872} C_VEL
LIN {X 0,Y 191.355,Z 492.647,A -85,B 0,C 180,E1 -21936.027,E2 -21936.027} C_VEL
LIN {X 0,Y 193.799,Z 507.565,A -85,B 0,C 180,E1 -21937.758,E2 -21937.758} C_VEL
LIN {X 0,Y 195.931,Z 519.805,A -85,B 0,C 180,E1 -21939.528,E2 -21939.528} C_VEL
LIN {X 0,Y 196.171,Z 523.3,A -85,B 0,C 180,E1 -21940.101,E2 -21940.101} C_VEL
LIN {X 0,Y 194.809,Z 534.385,A -85,B 0,C 180,E1 -21942.142,E2 -21942.142} C_VEL
LIN {X 0,Y 193.471,Z 545.831,A -85,B 0,C 180,E1 -21944.73,E2 -21944.73} C_VEL
LIN {X 0,Y 192.458,Z 555.365,A -85,B 0,C 180,E1 -21947.343,E2 -21947.343} C_VEL
LIN {X 0,Y 191.491,Z 564.73,A -85,B 0,C 180,E1 -21950.493,E2 -21950.493} C_VEL
LIN {X 0,Y 190.866,Z 572.867,A -85,B 0,C 180,E1 -21953.82,E2 -21953.82} C_VEL
LIN {X 0,Y 190.69,Z 578.934,A -85,B 0,C 180,E1 -21956.83,E2 -21956.83} C_VEL
LIN {X 0,Y 190.612,Z 584.127,A -85,B 0,C 180,E1 -21959.999,E2 -21959.999} C_VEL
LIN {X 0,Y 190.914,Z 588.294,A -85,B 0,C 180,E1 -21963.165,E2 -21963.165} C_VEL
LIN {X 0,Y 191.433,Z 591.565,A -85,B 0,C 180,E1 -21966.323,E2 -21966.323} C_VEL
LIN {X 0,Y 192.926,Z 594.669,A -85,B 0,C 180,E1 -21970.494,E2 -21970.494} C_VEL
LIN {X 0,Y 195.572,Z 596.378,A -85,B 0,C 180,E1 -21974.569,E2 -21974.569} C_VEL
LIN {X 0,Y 199.127,Z 596.768,A -85,B 0,C 180,E1 -21978.52,E2 -21978.52} C_VEL
LIN {X 0,Y 203.821,Z 595.871,A -85,B 0,C 180,E1 -21982.29,E2 -21982.29} C_VEL
LIN {X 0,Y 209.584,Z 593.647,A -85,B 0,C 180,E1 -21985.844,E2 -21985.844} C_VEL
LIN {X 0,Y 216.219,Z 590.109,A -85,B 0,C 180,E1 -21989.18,E2 -21989.18} C_VEL
LIN {X 0,Y 223.82,Z 585.186,A -85,B 0,C 180,E1 -21992.263,E2 -21992.263} C_VEL
LIN {X 0,Y 232.203,Z 578.7,A -85,B 0,C 180,E1 -21995.104,E2 -21995.104} C_VEL
LIN {X 0,Y 234.65,Z 576.644,A -85,B 0,C 180,E1 -21995.841,E2 -21995.841} C_VEL
LIN {X 0,Y 235.543,Z 575.554,A -85,B 0,C 180,E1 -21996.637,E2 -21996.637} C_VEL
LIN {X 0,Y 236.653,Z 573.914,A -85,B 0,C 180,E1 -21998.583,E2 -21998.583} C_VEL
LIN {X 0,Y 237.169,Z 573.022,A -85,B 0,C 180,E1 -22000.686,E2 -22000.686} C_VEL
LIN {X 0,Y 237.42,Z 572.835,A -85,B 0,C 180,E1 -22002.909,E2 -22002.909} C_VEL
LIN {X 0,Y 237.336,Z 573.571,A -85,B 0,C 180,E1 -22005.291,E2 -22005.291} C_VEL
LIN {X 0,Y 236.874,Z 574.842,A -85,B 0,C 180,E1 -22006.968,E2 -22006.968} C_VEL
LIN {X 0,Y 235.818,Z 576.494,A -85,B 0,C 180,E1 -22008.165,E2 -22008.165} C_VEL
LIN {X 0,Y 231.886,Z 581.381,A -85,B 0,C 180,E1 -22010.471,E2 -22010.471} C_VEL
LIN {X 0,Y 225.582,Z 588.602,A -85,B 0,C 180,E1 -22013.705,E2 -22013.705} C_VEL
LIN {X 0,Y 220.055,Z 593.889,A -85,B 0,C 180,E1 -22016.02,E2 -22016.02} C_VEL
LIN {X 0,Y 212.458,Z 600.019,A -85,B 0,C 180,E1 -22019.154,E2 -22019.154} C_VEL
LIN {X 0,Y 205.73,Z 604.916,A -85,B 0,C 180,E1 -22022.647,E2 -22022.647} C_VEL
LIN {X 0,Y 201.693,Z 607.543,A -85,B 0,C 180,E1 -22025.283,E2 -22025.283} C_VEL
LIN {X 0,Y 197.213,Z 610.136,A -85,B 0,C 180,E1 -22029.123,E2 -22029.123} C_VEL
LIN {X 0,Y 193.746,Z 611.512,A -85,B 0,C 180,E1 -22033.21,E2 -22033.21} C_VEL
LIN {X 0,Y 191.758,Z 611.62,A -85,B 0,C 180,E1 -22037.297,E2 -22037.297} C_VEL
LIN {X 0,Y 190.881,Z 610.444,A -85,B 0,C 180,E1 -22041.531,E2 -22041.531} C_VEL
LIN {X 0,Y 190.847,Z 610.031,A -85,B 0,C 180,E1 -22042.349,E2 -22042.349} C_VEL
LIN {X 0,Y 190.186,Z 609.339,A -85,B 0,C 180,E1 -22043.503,E2 -22043.503} C_VEL
LIN {X 0,Y 187.506,Z 607.57,A -85,B 0,C 180,E1 -22045.301,E2 -22045.301} C_VEL
LIN {X 0,Y 184.98,Z 605.443,A -85,B 0,C 180,E1 -22047.125,E2 -22047.125} C_VEL
LIN {X 0,Y 184.603,Z 604.136,A -85,B 0,C 180,E1 -22048.299,E2 -22048.299} C_VEL
LIN {X 0,Y 184.934,Z 603.098,A -85,B 0,C 180,E1 -22049.456,E2 -22049.456} C_VEL
LIN {X 0,Y 184.393,Z 606.084,A -85,B 0,C 180,E1 -22052.184,E2 -22052.184} C_VEL
LIN {X 0,Y 183.851,Z 609.538,A -85,B 0,C 180,E1 -22056.585,E2 -22056.585} C_VEL
LIN {X 0,Y 184.221,Z 611.551,A -85,B 0,C 180,E1 -22060.997,E2 -22060.997} C_VEL
LIN {X 0,Y 185.683,Z 612.318,A -85,B 0,C 180,E1 -22065.364,E2 -22065.364} C_VEL
LIN {X 0,Y 188.641,Z 611.894,A -85,B 0,C 180,E1 -22069.591,E2 -22069.591} C_VEL
LIN {X 0,Y 192.733,Z 610.275,A -85,B 0,C 180,E1 -22073.648,E2 -22073.648} C_VEL
LIN {X 0,Y 197.959,Z 607.483,A -85,B 0,C 180,E1 -22077.486,E2 -22077.486} C_VEL
LIN {X 0,Y 204.556,Z 603.517,A -85,B 0,C 180,E1 -22081.022,E2 -22081.022} C_VEL
LIN {X 0,Y 212.216,Z 598.253,A -85,B 0,C 180,E1 -22084.263,E2 -22084.263} C_VEL
LIN {X 0,Y 218.44,Z 593.466,A -85,B 0,C 180,E1 -22086.528,E2 -22086.528} C_VEL
LIN {X 0,Y 220.238,Z 591.825,A -85,B 0,C 180,E1 -22087.323,E2 -22087.323} C_VEL
LIN {X 0,Y 224.416,Z 587.233,A -85,B 0,C 180,E1 -22089.941,E2 -22089.941} C_VEL
LIN {X 0,Y 227.245,Z 583.899,A -85,B 0,C 180,E1 -22092.077,E2 -22092.077} C_VEL
LIN {X 0,Y 227.888,Z 583.043,A -85,B 0,C 180,E1 -22092.725,E2 -22092.725} C_VEL
LIN {X 0,Y 229.28,Z 580.9,A -85,B 0,C 180,E1 -22095.17,E2 -22095.17} C_VEL
LIN {X 0,Y 229.659,Z 580.003,A -85,B 0,C 180,E1 -22097.682,E2 -22097.682} C_VEL
LIN {X 0,Y 229.242,Z 580.235,A -85,B 0,C 180,E1 -22100.035,E2 -22100.035} C_VEL
LIN {X 0,Y 228.384,Z 581.49,A -85,B 0,C 180,E1 -22103.139,E2 -22103.139} C_VEL
LIN {X 0,Y 227.118,Z 582.544,A -85,B 0,C 180,E1 -22103.989,E2 -22103.989} C_VEL
LIN {X 0,Y 218.403,Z 588.421,A -85,B 0,C 180,E1 -22106.836,E2 -22106.836} C_VEL
LIN {X 0,Y 210.49,Z 592.804,A -85,B 0,C 180,E1 -22109.945,E2 -22109.945} C_VEL
LIN {X 0,Y 203.561,Z 595.857,A -85,B 0,C 180,E1 -22113.332,E2 -22113.332} C_VEL
LIN {X 0,Y 197.564,Z 597.664,A -85,B 0,C 180,E1 -22116.965,E2 -22116.965} C_VEL
LIN {X 0,Y 192.661,Z 598.199,A -85,B 0,C 180,E1 -22120.834,E2 -22120.834} C_VEL
LIN {X 0,Y 188.88,Z 597.443,A -85,B 0,C 180,E1 -22124.903,E2 -22124.903} C_VEL
LIN {X 0,Y 186.02,Z 595.402,A -85,B 0,C 180,E1 -22129.112,E2 -22129.112} C_VEL
LIN {X 0,Y 184.509,Z 592.044,A -85,B 0,C 180,E1 -22133.439,E2 -22133.439} C_VEL
LIN {X 0,Y 183.886,Z 588.575,A -85,B 0,C 180,E1 -22136.714,E2 -22136.714} C_VEL
LIN {X 0,Y 183.589,Z 582.514,A -85,B 0,C 180,E1 -22141.097,E2 -22141.097} C_VEL
LIN {X 0,Y 183.728,Z 575.425,A -85,B 0,C 180,E1 -22145.053,E2 -22145.053} C_VEL
LIN {X 0,Y 184.225,Z 568.393,A -85,B 0,C 180,E1 -22148.225,E2 -22148.225} C_VEL
LIN {X 0,Y 184.978,Z 559.581,A -85,B 0,C 180,E1 -22151.506,E2 -22151.506} C_VEL
LIN {X 0,Y 186.15,Z 548.826,A -85,B 0,C 180,E1 -22154.765,E2 -22154.765} C_VEL
LIN {X 0,Y 187.411,Z 538.008,A -85,B 0,C 180,E1 -22157.458,E2 -22157.458} C_VEL
LIN {X 0,Y 188.744,Z 527.599,A -85,B 0,C 180,E1 -22159.581,E2 -22159.581} C_VEL
LIN {X 0,Y 189.242,Z 522.461,A -85,B 0,C 180,E1 -22160.486,E2 -22160.486} C_VEL
LIN {X 0,Y 186.81,Z 508.825,A -85,B 0,C 180,E1 -22162.597,E2 -22162.597} C_VEL
LIN {X 0,Y 184.39,Z 493.997,A -85,B 0,C 180,E1 -22164.397,E2 -22164.397} C_VEL
LIN {X 0,Y 184.338,Z 493.524,A -85,B 0,C 180,E1 -22164.533,E2 -22164.533} C_VEL
LIN {X 0,Y 184.707,Z 493.476,A -85,B 0,C 180,E1 -22169.647,E2 -22169.647} C_VEL
LIN {X 0,Y 185.111,Z 493.421,A -85,B 0,C 180,E1 -22173.357,E2 -22173.357} C_VEL
LIN {X 0,Y 185.369,Z 493.393,A -85,B 0,C 180,E1 -22177.346,E2 -22177.346} C_VEL
LIN {X 0,Y 185.46,Z 493.379,A -85,B 0,C 180,E1 -22180.72,E2 -22180.72} C_VEL
LIN {X 0,Y 185.482,Z 493.381,A -85,B 0,C 180,E1 -22186.049,E2 -22186.049} C_VEL
LIN {X 0,Y 185.493,Z 493.376,A -85,B 0,C 180,E1 -22189.901,E2 -22189.901} C_VEL
LIN {X 0,Y 185.547,Z 493.371,A -85,B 0,C 180,E1 -22192.696,E2 -22192.696} C_VEL
LIN {X 0,Y 185.549,Z 493.371,A -85,B 0,C 180,E1 -22197.976,E2 -22197.976} C_VEL
LIN {X 0,Y 185.586,Z 493.366,A -85,B 0,C 180,E1 -22200.576,E2 -22200.576} C_VEL
LIN {X 0,Y 185.591,Z 493.365,A -85,B 0,C 180,E1 -22205.383,E2 -22205.383} C_VEL
LIN {X 0,Y 185.611,Z 493.363,A -85,B 0,C 180,E1 -22210.076,E2 -22210.076} C_VEL
LIN {X 0,Y 185.729,Z 493.347,A -85,B 0,C 180,E1 -22214.64,E2 -22214.64} C_VEL
LIN {X 0,Y 185.947,Z 493.32,A -85,B 0,C 180,E1 -22219.328,E2 -22219.328} C_VEL
LIN {X 0,Y 185.974,Z 493.318,A -85,B 0,C 180,E1 -22223.49,E2 -22223.49} C_VEL
LIN {X 0,Y 186.213,Z 493.288,A -85,B 0,C 180,E1 -22227.837,E2 -22227.837} C_VEL
LIN {X 0,Y 186.411,Z 493.266,A -85,B 0,C 180,E1 -22230,E2 -22230} C_VEL
LIN {X 0,Y 185.918,Z 493.322,A -85,B 0,C 180,E1 -22234.336,E2 -22234.336} C_VEL
LIN {X 0,Y 185.983,Z 493.317,A -85,B 0,C 180,E1 -22238.694,E2 -22238.694} C_VEL
LIN {X 0,Y 185.736,Z 493.343,A -85,B 0,C 180,E1 -22243.122,E2 -22243.122} C_VEL
LIN {X 0,Y 185.695,Z 493.354,A -85,B 0,C 180,E1 -22247.625,E2 -22247.625} C_VEL
LIN {X 0,Y 185.601,Z 493.362,A -85,B 0,C 180,E1 -22252.251,E2 -22252.251} C_VEL
LIN {X 0,Y 185.567,Z 493.369,A -85,B 0,C 180,E1 -22257.032,E2 -22257.032} C_VEL
LIN {X 0,Y 185.583,Z 493.366,A -85,B 0,C 180,E1 -22259.493,E2 -22259.493} C_VEL
LIN {X 0,Y 185.523,Z 493.374,A -85,B 0,C 180,E1 -22264.627,E2 -22264.627} C_VEL
LIN {X 0,Y 185.547,Z 493.371,A -85,B 0,C 180,E1 -22267.304,E2 -22267.304} C_VEL
LIN {X 0,Y 185.489,Z 493.375,A -85,B 0,C 180,E1 -22270.73,E2 -22270.73} C_VEL
LIN {X 0,Y 185.482,Z 493.381,A -85,B 0,C 180,E1 -22273.951,E2 -22273.951} C_VEL
LIN {X 0,Y 185.467,Z 493.378,A -85,B 0,C 180,E1 -22279.277,E2 -22279.277} C_VEL
LIN {X 0,Y 185.447,Z 493.383,A -85,B 0,C 180,E1 -22282.736,E2 -22282.736} C_VEL
LIN {X 0,Y 185.191,Z 493.411,A -85,B 0,C 180,E1 -22286.606,E2 -22286.606} C_VEL
LIN {X 0,Y 184.769,Z 493.468,A -85,B 0,C 180,E1 -22291.027,E2 -22291.027} C_VEL
LIN {X 0,Y 184.315,Z 493.523,A -85,B 0,C 180,E1 -22295.922,E2 -22295.922} C_VEL
LIN {X 0,Y 186.761,Z 508.477,A -85,B 0,C 180,E1 -22297.749,E2 -22297.749} C_VEL
LIN {X 0,Y 189.123,Z 521.971,A -85,B 0,C 180,E1 -22299.823,E2 -22299.823} C_VEL
LIN {X 0,Y 187.983,Z 532.398,A -85,B 0,C 180,E1 -22301.753,E2 -22301.753} C_VEL
LIN {X 0,Y 186.678,Z 543.081,A -85,B 0,C 180,E1 -22304.16,E2 -22304.16} C_VEL
LIN {X 0,Y 185.386,Z 554.78,A -85,B 0,C 180,E1 -22307.409,E2 -22307.409} C_VEL
LIN {X 0,Y 184.399,Z 564.355,A -85,B 0,C 180,E1 -22310.678,E2 -22310.678} C_VEL
LIN {X 0,Y 183.784,Z 572.66,A -85,B 0,C 180,E1 -22314.152,E2 -22314.152} C_VEL
LIN {X 0,Y 183.606,Z 579.695,A -85,B 0,C 180,E1 -22317.806,E2 -22317.806} C_VEL
LIN {X 0,Y 183.71,Z 586.273,A -85,B 0,C 180,E1 -22322.192,E2 -22322.192} C_VEL
LIN {X 0,Y 184.194,Z 590.093,A -85,B 0,C 180,E1 -22325.473,E2 -22325.473} C_VEL
LIN {X 0,Y 185.403,Z 593.806,A -85,B 0,C 180,E1 -22329.743,E2 -22329.743} C_VEL
LIN {X 0,Y 187.226,Z 595.78,A -85,B 0,C 180,E1 -22333.016,E2 -22333.016} C_VEL
LIN {X 0,Y 190.361,Z 597.21,A -85,B 0,C 180,E1 -22337.178,E2 -22337.178} C_VEL
LIN {X 0,Y 194.882,Z 597.325,A -85,B 0,C 180,E1 -22341.138,E2 -22341.138} C_VEL
LIN {X 0,Y 200.221,Z 596.157,A -85,B 0,C 180,E1 -22344.911,E2 -22344.911} C_VEL
LIN {X 0,Y 206.691,Z 593.711,A -85,B 0,C 180,E1 -22348.426,E2 -22348.426} C_VEL
LIN {X 0,Y 214.076,Z 590.007,A -85,B 0,C 180,E1 -22351.686,E2 -22351.686} C_VEL
LIN {X 0,Y 222.367,Z 584.837,A -85,B 0,C 180,E1 -22354.673,E2 -22354.673} C_VEL
LIN {X 0,Y 228.839,Z 580.169,A -85,B 0,C 180,E1 -22356.669,E2 -22356.669} C_VEL
LIN {X 0,Y 230.179,Z 578.954,A -85,B 0,C 180,E1 -22357.637,E2 -22357.637} C_VEL
LIN {X 0,Y 231.265,Z 577.679,A -85,B 0,C 180,E1 -22359.656,E2 -22359.656} C_VEL
LIN {X 0,Y 231.705,Z 577.216,A -85,B 0,C 180,E1 -22361.859,E2 -22361.859} C_VEL
LIN {X 0,Y 231.806,Z 577.554,A -85,B 0,C 180,E1 -22364.213,E2 -22364.213} C_VEL
LIN {X 0,Y 231.537,Z 578.338,A -85,B 0,C 180,E1 -22365.722,E2 -22365.722} C_VEL
LIN {X 0,Y 230.912,Z 579.4,A -85,B 0,C 180,E1 -22366.925,E2 -22366.925} C_VEL
LIN {X 0,Y 229.895,Z 580.645,A -85,B 0,C 180,E1 -22367.736,E2 -22367.736} C_VEL
LIN {X 0,Y 225.177,Z 585.644,A -85,B 0,C 180,E1 -22370.221,E2 -22370.221} C_VEL
LIN {X 0,Y 218.32,Z 592.264,A -85,B 0,C 180,E1 -22373.449,E2 -22373.449} C_VEL
LIN {X 0,Y 210.295,Z 598.432,A -85,B 0,C 180,E1 -22376.535,E2 -22376.535} C_VEL
LIN {X 0,Y 202.912,Z 603.37,A -85,B 0,C 180,E1 -22379.853,E2 -22379.853} C_VEL
LIN {X 0,Y 198.035,Z 606.279,A -85,B 0,C 180,E1 -22382.525,E2 -22382.525} C_VEL
LIN {X 0,Y 192.804,Z 609.054,A -85,B 0,C 180,E1 -22386.361,E2 -22386.361} C_VEL
LIN {X 0,Y 188.693,Z 610.657,A -85,B 0,C 180,E1 -22390.415,E2 -22390.415} C_VEL
LIN {X 0,Y 185.673,Z 611.042,A -85,B 0,C 180,E1 -22394.635,E2 -22394.635} C_VEL
LIN {X 0,Y 184.218,Z 610.231,A -85,B 0,C 180,E1 -22399.003,E2 -22399.003} C_VEL
LIN {X 0,Y 183.915,Z 608.111,A -85,B 0,C 180,E1 -22403.485,E2 -22403.485} C_VEL
LIN {X 0,Y 184.474,Z 604.616,A -85,B 0,C 180,E1 -22407.817,E2 -22407.817} C_VEL
LIN {X 0,Y 184.603,Z 604.136,A -85,B 0,C 180,E1 -22408.299,E2 -22408.299} C_VEL
LIN {X 0,Y 184.47,Z 603.73,A -85,B 0,C 180,E1 -22409.473,E2 -22409.473} C_VEL
LIN {X 0,Y 183.685,Z 604.251,A -85,B 0,C 180,E1 -22410.648,E2 -22410.648} C_VEL
LIN {X 0,Y 181.051,Z 606.055,A -85,B 0,C 180,E1 -22412.966,E2 -22412.966} C_VEL
LIN {X 0,Y 178.213,Z 607.529,A -85,B 0,C 180,E1 -22415.379,E2 -22415.379} C_VEL
LIN {X 0,Y 176.986,Z 608.475,A -85,B 0,C 180,E1 -22417.287,E2 -22417.287} C_VEL
LIN {X 0,Y 176.902,Z 608.795,A -85,B 0,C 180,E1 -22417.936,E2 -22417.936} C_VEL
LIN {X 0,Y 177.318,Z 610.494,A -85,B 0,C 180,E1 -22421.43,E2 -22421.43} C_VEL
LIN {X 0,Y 178.854,Z 611.561,A -85,B 0,C 180,E1 -22425.966,E2 -22425.966} C_VEL
LIN {X 0,Y 181.961,Z 611.491,A -85,B 0,C 180,E1 -22430.341,E2 -22430.341} C_VEL
LIN {X 0,Y 186.245,Z 610.238,A -85,B 0,C 180,E1 -22434.525,E2 -22434.525} C_VEL
LIN {X 0,Y 191.7,Z 607.85,A -85,B 0,C 180,E1 -22438.464,E2 -22438.464} C_VEL
LIN {X 0,Y 198.552,Z 604.28,A -85,B 0,C 180,E1 -22442.069,E2 -22442.069} C_VEL
LIN {X 0,Y 206.478,Z 599.519,A -85,B 0,C 180,E1 -22445.355,E2 -22445.355} C_VEL
LIN {X 0,Y 212.916,Z 595.187,A -85,B 0,C 180,E1 -22447.637,E2 -22447.637} C_VEL
LIN {X 0,Y 214.794,Z 593.675,A -85,B 0,C 180,E1 -22448.439,E2 -22448.439} C_VEL
LIN {X 0,Y 219.191,Z 589.499,A -85,B 0,C 180,E1 -22451.094,E2 -22451.094} C_VEL
LIN {X 0,Y 222.056,Z 586.497,A -85,B 0,C 180,E1 -22453.286,E2 -22453.286} C_VEL
LIN {X 0,Y 223.557,Z 584.389,A -85,B 0,C 180,E1 -22456.308,E2 -22456.308} C_VEL
LIN {X 0,Y 223.443,Z 584.019,A -85,B 0,C 180,E1 -22459.015,E2 -22459.015} C_VEL
LIN {X 0,Y 222.632,Z 584.767,A -85,B 0,C 180,E1 -22462.111,E2 -22462.111} C_VEL
LIN {X 0,Y 221.744,Z 585.46,A -85,B 0,C 180,E1 -22462.973,E2 -22462.973} C_VEL
LIN {X 0,Y 212.759,Z 590.707,A -85,B 0,C 180,E1 -22465.837,E2 -22465.837} C_VEL
LIN {X 0,Y 204.581,Z 594.655,A -85,B 0,C 180,E1 -22468.983,E2 -22468.983} C_VEL
LIN {X 0,Y 197.371,Z 597.247,A -85,B 0,C 180,E1 -22472.426,E2 -22472.426} C_VEL
LIN {X 0,Y 191.122,Z 598.603,A -85,B 0,C 180,E1 -22476.141,E2 -22476.141} C_VEL
LIN {X 0,Y 186.002,Z 598.753,A -85,B 0,C 180,E1 -22480.12,E2 -22480.12} C_VEL
LIN {X 0,Y 182.056,Z 597.652,A -85,B 0,C 180,E1 -22484.323,E2 -22484.323} C_VEL
LIN {X 0,Y 179.068,Z 595.268,A -85,B 0,C 180,E1 -22488.683,E2 -22488.683} C_VEL
LIN {X 0,Y 177.499,Z 591.55,A -85,B 0,C 180,E1 -22493.179,E2 -22493.179} C_VEL
LIN {X 0,Y 176.835,Z 587.835,A -85,B 0,C 180,E1 -22496.583,E2 -22496.583} C_VEL
LIN {X 0,Y 176.528,Z 583.221,A -85,B 0,C 180,E1 -22500.001,E2 -22500.001} C_VEL
LIN {X 0,Y 176.64,Z 576.421,A -85,B 0,C 180,E1 -22503.993,E2 -22503.993} C_VEL
LIN {X 0,Y 177.168,Z 567.998,A -85,B 0,C 180,E1 -22507.981,E2 -22507.981} C_VEL
LIN {X 0,Y 177.892,Z 559.073,A -85,B 0,C 180,E1 -22511.394,E2 -22511.394} C_VEL
LIN {X 0,Y 178.84,Z 550.108,A -85,B 0,C 180,E1 -22514.219,E2 -22514.219} C_VEL
LIN {X 0,Y 180.173,Z 539.495,A -85,B 0,C 180,E1 -22517.011,E2 -22517.011} C_VEL
LIN {X 0,Y 181.578,Z 527.946,A -85,B 0,C 180,E1 -22519.502,E2 -22519.502} C_VEL
LIN {X 0,Y 182.05,Z 523.522,A -85,B 0,C 180,E1 -22520.332,E2 -22520.332} C_VEL
LIN {X 0,Y 180.384,Z 513.287,A -85,B 0,C 180,E1 -22522.029,E2 -22522.029} C_VEL
LIN {X 0,Y 177.995,Z 498.655,A -85,B 0,C 180,E1 -22524.016,E2 -22524.016} C_VEL
LIN {X 0,Y 177.298,Z 494.401,A -85,B 0,C 180,E1 -22524.511,E2 -22524.511} C_VEL
LIN {X 0,Y 177.645,Z 494.355,A -85,B 0,C 180,E1 -22529.499,E2 -22529.499} C_VEL
LIN {X 0,Y 178.095,Z 494.296,A -85,B 0,C 180,E1 -22534.034,E2 -22534.034} C_VEL
LIN {X 0,Y 178.347,Z 494.267,A -85,B 0,C 180,E1 -22539.088,E2 -22539.088} C_VEL
LIN {X 0,Y 178.396,Z 494.259,A -85,B 0,C 180,E1 -22542.047,E2 -22542.047} C_VEL
LIN {X 0,Y 178.404,Z 494.261,A -85,B 0,C 180,E1 -22545.162,E2 -22545.162} C_VEL
LIN {X 0,Y 178.414,Z 494.259,A -85,B 0,C 180,E1 -22548.457,E2 -22548.457} C_VEL
LIN {X 0,Y 178.467,Z 494.251,A -85,B 0,C 180,E1 -22551.963,E2 -22551.963} C_VEL
LIN {X 0,Y 178.495,Z 494.249,A -85,B 0,C 180,E1 -22556.548,E2 -22556.548} C_VEL
LIN {X 0,Y 178.526,Z 494.242,A -85,B 0,C 180,E1 -22560.007,E2 -22560.007} C_VEL
LIN {X 0,Y 178.538,Z 494.244,A -85,B 0,C 180,E1 -22564.876,E2 -22564.876} C_VEL
LIN {X 0,Y 178.627,Z 494.233,A -85,B 0,C 180,E1 -22570.784,E2 -22570.784} C_VEL
LIN {X 0,Y 178.67,Z 494.229,A -85,B 0,C 180,E1 -22574.017,E2 -22574.017} C_VEL
LIN {X 0,Y 178.899,Z 494.198,A -85,B 0,C 180,E1 -22579.153,E2 -22579.153} C_VEL
LIN {X 0,Y 178.939,Z 494.193,A -85,B 0,C 180,E1 -22583.233,E2 -22583.233} C_VEL
LIN {X 0,Y 179.159,Z 494.166,A -85,B 0,C 180,E1 -22587.752,E2 -22587.752} C_VEL
LIN {X 0,Y 179.374,Z 494.143,A -85,B 0,C 180,E1 -22590,E2 -22590} C_VEL
LIN {X 0,Y 178.866,Z 494.2,A -85,B 0,C 180,E1 -22594.507,E2 -22594.507} C_VEL
LIN {X 0,Y 178.912,Z 494.198,A -85,B 0,C 180,E1 -22599.04,E2 -22599.04} C_VEL
LIN {X 0,Y 178.663,Z 494.225,A -85,B 0,C 180,E1 -22603.652,E2 -22603.652} C_VEL
LIN {X 0,Y 178.627,Z 494.233,A -85,B 0,C 180,E1 -22609.216,E2 -22609.216} C_VEL
LIN {X 0,Y 178.538,Z 494.244,A -85,B 0,C 180,E1 -22615.124,E2 -22615.124} C_VEL
LIN {X 0,Y 178.483,Z 494.246,A -85,B 0,C 180,E1 -22620.79,E2 -22620.79} C_VEL
LIN {X 0,Y 178.5,Z 494.25,A -85,B 0,C 180,E1 -22624.225,E2 -22624.225} C_VEL
LIN {X 0,Y 178.422,Z 494.255,A -85,B 0,C 180,E1 -22629.068,E2 -22629.068} C_VEL
LIN {X 0,Y 178.406,Z 494.262,A -85,B 0,C 180,E1 -22632.043,E2 -22632.043} C_VEL
LIN {X 0,Y 178.401,Z 494.262,A -85,B 0,C 180,E1 -22635.162,E2 -22635.162} C_VEL
LIN {X 0,Y 178.403,Z 494.257,A -85,B 0,C 180,E1 -22638.46,E2 -22638.46} C_VEL
LIN {X 0,Y 178.374,Z 494.266,A -85,B 0,C 180,E1 -22642,E2 -22642} C_VEL
LIN {X 0,Y 178.173,Z 494.285,A -85,B 0,C 180,E1 -22646.479,E2 -22646.479} C_VEL
LIN {X 0,Y 177.625,Z 494.361,A -85,B 0,C 180,E1 -22651.653,E2 -22651.653} C_VEL
LIN {X 0,Y 177.277,Z 494.428,A -85,B 0,C 180,E1 -22655.914,E2 -22655.914} C_VEL
LIN {X 0,Y 179.639,Z 508.819,A -85,B 0,C 180,E1 -22657.726,E2 -22657.726} C_VEL
LIN {X 0,Y 181.768,Z 520.983,A -85,B 0,C 180,E1 -22659.635,E2 -22659.635} C_VEL
LIN {X 0,Y 181.987,Z 522.784,A -85,B 0,C 180,E1 -22659.956,E2 -22659.956} C_VEL
LIN {X 0,Y 180.596,Z 533.938,A -85,B 0,C 180,E1 -22662.153,E2 -22662.153} C_VEL
LIN {X 0,Y 179.37,Z 544.428,A -85,B 0,C 180,E1 -22664.664,E2 -22664.664} C_VEL
LIN {X 0,Y 178.111,Z 555.97,A -85,B 0,C 180,E1 -22668.044,E2 -22668.044} C_VEL
LIN {X 0,Y 177.246,Z 565.325,A -85,B 0,C 180,E1 -22671.448,E2 -22671.448} C_VEL
LIN {X 0,Y 176.645,Z 574.2,A -85,B 0,C 180,E1 -22675.435,E2 -22675.435} C_VEL
LIN {X 0,Y 176.541,Z 580.4,A -85,B 0,C 180,E1 -22678.859,E2 -22678.859} C_VEL
LIN {X 0,Y 176.656,Z 585.441,A -85,B 0,C 180,E1 -22682.279,E2 -22682.279} C_VEL
LIN {X 0,Y 177.166,Z 589.496,A -85,B 0,C 180,E1 -22685.691,E2 -22685.691} C_VEL
LIN {X 0,Y 178.192,Z 593.122,A -85,B 0,C 180,E1 -22689.591,E2 -22689.591} C_VEL
LIN {X 0,Y 180.316,Z 595.792,A -85,B 0,C 180,E1 -22693.524,E2 -22693.524} C_VEL
LIN {X 0,Y 183.619,Z 597.57,A -85,B 0,C 180,E1 -22697.83,E2 -22697.83} C_VEL
LIN {X 0,Y 188.325,Z 598.039,A -85,B 0,C 180,E1 -22701.912,E2 -22701.912} C_VEL
LIN {X 0,Y 193.888,Z 597.301,A -85,B 0,C 180,E1 -22705.783,E2 -22705.783} C_VEL
LIN {X 0,Y 200.627,Z 595.321,A -85,B 0,C 180,E1 -22709.368,E2 -22709.368} C_VEL
LIN {X 0,Y 208.28,Z 592.055,A -85,B 0,C 180,E1 -22712.676,E2 -22712.676} C_VEL
LIN {X 0,Y 216.857,Z 587.41,A -85,B 0,C 180,E1 -22715.686,E2 -22715.686} C_VEL
LIN {X 0,Y 223.934,Z 582.943,A -85,B 0,C 180,E1 -22717.81,E2 -22717.81} C_VEL
LIN {X 0,Y 224.708,Z 582.268,A -85,B 0,C 180,E1 -22718.72,E2 -22718.72} C_VEL
LIN {X 0,Y 225.732,Z 581.427,A -85,B 0,C 180,E1 -22720.83,E2 -22720.83} C_VEL
LIN {X 0,Y 226.035,Z 581.441,A -85,B 0,C 180,E1 -22723.16,E2 -22723.16} C_VEL
LIN {X 0,Y 225.962,Z 581.769,A -85,B 0,C 180,E1 -22724.327,E2 -22724.327} C_VEL
LIN {X 0,Y 225.562,Z 582.586,A -85,B 0,C 180,E1 -22725.777,E2 -22725.777} C_VEL
LIN {X 0,Y 224.928,Z 583.359,A -85,B 0,C 180,E1 -22726.575,E2 -22726.575} C_VEL
LIN {X 0,Y 221.765,Z 586.343,A -85,B 0,C 180,E1 -22728.278,E2 -22728.278} C_VEL
LIN {X 0,Y 214.724,Z 592.465,A -85,B 0,C 180,E1 -22731.547,E2 -22731.547} C_VEL
LIN {X 0,Y 208.656,Z 596.948,A -85,B 0,C 180,E1 -22733.883,E2 -22733.883} C_VEL
LIN {X 0,Y 200.535,Z 602.012,A -85,B 0,C 180,E1 -22737.097,E2 -22737.097} C_VEL
LIN {X 0,Y 195.163,Z 605.001,A -85,B 0,C 180,E1 -22739.725,E2 -22739.725} C_VEL
LIN {X 0,Y 191.261,Z 606.901,A -85,B 0,C 180,E1 -22741.871,E2 -22741.871} C_VEL
LIN {X 0,Y 186.316,Z 609.035,A -85,B 0,C 180,E1 -22745.485,E2 -22745.485} C_VEL
LIN {X 0,Y 182.028,Z 610.266,A -85,B 0,C 180,E1 -22749.666,E2 -22749.666} C_VEL
LIN {X 0,Y 178.845,Z 610.289,A -85,B 0,C 180,E1 -22754.033,E2 -22754.033} C_VEL
LIN {X 0,Y 177.315,Z 609.166,A -85,B 0,C 180,E1 -22758.569,E2 -22758.569} C_VEL
LIN {X 0,Y 176.96,Z 606.786,A -85,B 0,C 180,E1 -22763.157,E2 -22763.157} C_VEL
LIN {X 0,Y 177.571,Z 602.99,A -85,B 0,C 180,E1 -22767.732,E2 -22767.732} C_VEL
LIN {X 0,Y 178.061,Z 601.262,A -85,B 0,C 180,E1 -22769.435,E2 -22769.435} C_VEL
LIN {X 0,Y 177.499,Z 604.455,A -85,B 0,C 180,E1 -22772.269,E2 -22772.269} C_VEL
LIN {X 0,Y 176.905,Z 608.168,A -85,B 0,C 180,E1 -22776.845,E2 -22776.845} C_VEL
LIN {X 0,Y 176.902,Z 608.795,A -85,B 0,C 180,E1 -22777.936,E2 -22777.936} C_VEL
LIN {X 0,Y 176.376,Z 609.699,A -85,B 0,C 180,E1 -22779.824,E2 -22779.824} C_VEL
LIN {X 0,Y 174.158,Z 610.41,A -85,B 0,C 180,E1 -22782.977,E2 -22782.977} C_VEL
LIN {X 0,Y 172.573,Z 610.736,A -85,B 0,C 180,E1 -22786.214,E2 -22786.214} C_VEL
LIN {X 0,Y 173.039,Z 610.879,A -85,B 0,C 180,E1 -22788.166,E2 -22788.166} C_VEL
LIN {X 0,Y 175.336,Z 610.945,A -85,B 0,C 180,E1 -22791.146,E2 -22791.146} C_VEL
LIN {X 0,Y 179.806,Z 610.053,A -85,B 0,C 180,E1 -22795.465,E2 -22795.465} C_VEL
LIN {X 0,Y 185.506,Z 608.059,A -85,B 0,C 180,E1 -22799.506,E2 -22799.506} C_VEL
LIN {X 0,Y 192.608,Z 604.957,A -85,B 0,C 180,E1 -22803.184,E2 -22803.184} C_VEL
LIN {X 0,Y 200.801,Z 600.685,A -85,B 0,C 180,E1 -22806.513,E2 -22806.513} C_VEL
LIN {X 0,Y 207.445,Z 596.741,A -85,B 0,C 180,E1 -22808.812,E2 -22808.812} C_VEL
LIN {X 0,Y 209.398,Z 595.348,A -85,B 0,C 180,E1 -22809.62,E2 -22809.62} C_VEL
LIN {X 0,Y 212.547,Z 592.83,A -85,B 0,C 180,E1 -22811.4,E2 -22811.4} C_VEL
LIN {X 0,Y 215.31,Z 590.419,A -85,B 0,C 180,E1 -22813.273,E2 -22813.273} C_VEL
LIN {X 0,Y 216.464,Z 589.294,A -85,B 0,C 180,E1 -22814.416,E2 -22814.416} C_VEL
LIN {X 0,Y 216.922,Z 588.639,A -85,B 0,C 180,E1 -22815.461,E2 -22815.461} C_VEL
LIN {X 0,Y 217.412,Z 587.903,A -85,B 0,C 180,E1 -22817.247,E2 -22817.247} C_VEL
LIN {X 0,Y 217.142,Z 587.765,A -85,B 0,C 180,E1 -22819.661,E2 -22819.661} C_VEL
LIN {X 0,Y 216.35,Z 588.258,A -85,B 0,C 180,E1 -22821.888,E2 -22821.888} C_VEL
LIN {X 0,Y 207.156,Z 592.946,A -85,B 0,C 180,E1 -22824.778,E2 -22824.778} C_VEL
LIN {X 0,Y 198.692,Z 596.365,A -85,B 0,C 180,E1 -22827.956,E2 -22827.956} C_VEL
LIN {X 0,Y 191.226,Z 598.521,A -85,B 0,C 180,E1 -22831.46,E2 -22831.46} C_VEL
LIN {X 0,Y 184.72,Z 599.478,A -85,B 0,C 180,E1 -22835.26,E2 -22835.26} C_VEL
LIN {X 0,Y 179.367,Z 599.209,A -85,B 0,C 180,E1 -22839.352,E2 -22839.352} C_VEL
LIN {X 0,Y 175.229,Z 597.718,A -85,B 0,C 180,E1 -22843.695,E2 -22843.695} C_VEL
LIN {X 0,Y 172.142,Z 594.983,A -85,B 0,C 180,E1 -22848.222,E2 -22848.222} C_VEL
LIN {X 0,Y 170.492,Z 590.975,A -85,B 0,C 180,E1 -22852.897,E2 -22852.897} C_VEL
LIN {X 0,Y 169.816,Z 586.963,A -85,B 0,C 180,E1 -22856.441,E2 -22856.441} C_VEL
LIN {X 0,Y 169.526,Z 582.037,A -85,B 0,C 180,E1 -22860.001,E2 -22860.001} C_VEL
LIN {X 0,Y 169.624,Z 576.089,A -85,B 0,C 180,E1 -22863.564,E2 -22863.564} C_VEL
LIN {X 0,Y 170.112,Z 567.606,A -85,B 0,C 180,E1 -22867.657,E2 -22867.657} C_VEL
LIN {X 0,Y 170.842,Z 558.37,A -85,B 0,C 180,E1 -22871.269,E2 -22871.269} C_VEL
LIN {X 0,Y 171.801,Z 549.367,A -85,B 0,C 180,E1 -22874.209,E2 -22874.209} C_VEL
LIN {X 0,Y 173.123,Z 538.619,A -85,B 0,C 180,E1 -22877.117,E2 -22877.117} C_VEL
LIN {X 0,Y 174.584,Z 526.776,A -85,B 0,C 180,E1 -22879.704,E2 -22879.704} C_VEL
LIN {X 0,Y 174.785,Z 522.025,A -85,B 0,C 180,E1 -22880.6,E2 -22880.6} C_VEL
LIN {X 0,Y 172.383,Z 508.595,A -85,B 0,C 180,E1 -22882.805,E2 -22882.805} C_VEL
LIN {X 0,Y 170.258,Z 495.277,A -85,B 0,C 180,E1 -22884.568,E2 -22884.568} C_VEL
LIN {X 0,Y 170.661,Z 495.227,A -85,B 0,C 180,E1 -22890.14,E2 -22890.14} C_VEL
LIN {X 0,Y 171.079,Z 495.172,A -85,B 0,C 180,E1 -22895.109,E2 -22895.109} C_VEL
LIN {X 0,Y 171.289,Z 495.147,A -85,B 0,C 180,E1 -22898.778,E2 -22898.778} C_VEL
LIN {X 0,Y 171.335,Z 495.139,A -85,B 0,C 180,E1 -22902.409,E2 -22902.409} C_VEL
LIN {X 0,Y 171.343,Z 495.14,A -85,B 0,C 180,E1 -22907.589,E2 -22907.589} C_VEL
LIN {X 0,Y 171.417,Z 495.129,A -85,B 0,C 180,E1 -22912.048,E2 -22912.048} C_VEL
LIN {X 0,Y 171.414,Z 495.132,A -85,B 0,C 180,E1 -22915.087,E2 -22915.087} C_VEL
LIN {X 0,Y 171.453,Z 495.126,A -85,B 0,C 180,E1 -22920.535,E2 -22920.535} C_VEL
LIN {X 0,Y 171.462,Z 495.126,A -85,B 0,C 180,E1 -22925.802,E2 -22925.802} C_VEL
LIN {X 0,Y 171.583,Z 495.11,A -85,B 0,C 180,E1 -22930.872,E2 -22930.872} C_VEL
LIN {X 0,Y 171.614,Z 495.106,A -85,B 0,C 180,E1 -22935.776,E2 -22935.776} C_VEL
LIN {X 0,Y 171.915,Z 495.07,A -85,B 0,C 180,E1 -22940.589,E2 -22940.589} C_VEL
LIN {X 0,Y 171.83,Z 495.076,A -85,B 0,C 180,E1 -22945.308,E2 -22945.308} C_VEL
LIN {X 0,Y 172.337,Z 495.02,A -85,B 0,C 180,E1 -22950,E2 -22950} C_VEL
LIN {X 0,Y 171.814,Z 495.078,A -85,B 0,C 180,E1 -22954.693,E2 -22954.693} C_VEL
LIN {X 0,Y 171.85,Z 495.078,A -85,B 0,C 180,E1 -22959.415,E2 -22959.415} C_VEL
LIN {X 0,Y 171.581,Z 495.11,A -85,B 0,C 180,E1 -22964.227,E2 -22964.227} C_VEL
LIN {X 0,Y 171.549,Z 495.116,A -85,B 0,C 180,E1 -22969.562,E2 -22969.562} C_VEL
LIN {X 0,Y 171.473,Z 495.125,A -85,B 0,C 180,E1 -22975.616,E2 -22975.616} C_VEL
LIN {X 0,Y 171.445,Z 495.122,A -85,B 0,C 180,E1 -22980.587,E2 -22980.587} C_VEL
LIN {X 0,Y 171.41,Z 495.132,A -85,B 0,C 180,E1 -22985.031,E2 -22985.031} C_VEL
LIN {X 0,Y 171.383,Z 495.131,A -85,B 0,C 180,E1 -22988.816,E2 -22988.816} C_VEL
LIN {X 0,Y 171.33,Z 495.143,A -85,B 0,C 180,E1 -22994.215,E2 -22994.215} C_VEL
LIN {X 0,Y 171.332,Z 495.137,A -85,B 0,C 180,E1 -22998.979,E2 -22998.979} C_VEL
LIN {X 0,Y 171.324,Z 495.144,A -85,B 0,C 180,E1 -23002.023,E2 -23002.023} C_VEL
LIN {X 0,Y 171.162,Z 495.163,A -85,B 0,C 180,E1 -23005.206,E2 -23005.206} C_VEL
LIN {X 0,Y 170.742,Z 495.215,A -85,B 0,C 180,E1 -23010.399,E2 -23010.399} C_VEL
LIN {X 0,Y 170.238,Z 495.276,A -85,B 0,C 180,E1 -23015.86,E2 -23015.86} C_VEL
LIN {X 0,Y 172.714,Z 510.355,A -85,B 0,C 180,E1 -23017.889,E2 -23017.889} C_VEL
LIN {X 0,Y 174.816,Z 523.038,A -85,B 0,C 180,E1 -23020.018,E2 -23020.018} C_VEL
LIN {X 0,Y 173.437,Z 534.21,A -85,B 0,C 180,E1 -23022.306,E2 -23022.306} C_VEL
LIN {X 0,Y 172.335,Z 543.615,A -85,B 0,C 180,E1 -23024.628,E2 -23024.628} C_VEL
LIN {X 0,Y 171.271,Z 553.457,A -85,B 0,C 180,E1 -23027.559,E2 -23027.559} C_VEL
LIN {X 0,Y 170.298,Z 563.26,A -85,B 0,C 180,E1 -23031.097,E2 -23031.097} C_VEL
LIN {X 0,Y 169.7,Z 571.628,A -85,B 0,C 180,E1 -23034.754,E2 -23034.754} C_VEL
LIN {X 0,Y 169.548,Z 578.132,A -85,B 0,C 180,E1 -23038.218,E2 -23038.218} C_VEL
LIN {X 0,Y 169.638,Z 584.413,A -85,B 0,C 180,E1 -23042.374,E2 -23042.374} C_VEL
LIN {X 0,Y 170.143,Z 588.779,A -85,B 0,C 180,E1 -23045.927,E2 -23045.927} C_VEL
LIN {X 0,Y 171.117,Z 592.442,A -85,B 0,C 180,E1 -23049.697,E2 -23049.697} C_VEL
LIN {X 0,Y 173.429,Z 595.657,A -85,B 0,C 180,E1 -23054.072,E2 -23054.072} C_VEL
LIN {X 0,Y 176.877,Z 597.788,A -85,B 0,C 180,E1 -23058.534,E2 -23058.534} C_VEL
LIN {X 0,Y 181.791,Z 598.675,A -85,B 0,C 180,E1 -23062.743,E2 -23062.743} C_VEL
LIN {X 0,Y 187.598,Z 598.356,A -85,B 0,C 180,E1 -23066.715,E2 -23066.715} C_VEL
LIN {X 0,Y 194.605,Z 596.782,A -85,B 0,C 180,E1 -23070.371,E2 -23070.371} C_VEL
LIN {X 0,Y 202.537,Z 593.995,A -85,B 0,C 180,E1 -23073.724,E2 -23073.724} C_VEL
LIN {X 0,Y 211.421,Z 589.911,A -85,B 0,C 180,E1 -23076.752,E2 -23076.752} C_VEL
LIN {X 0,Y 218.621,Z 585.895,A -85,B 0,C 180,E1 -23078.922,E2 -23078.922} C_VEL
LIN {X 0,Y 219.142,Z 585.566,A -85,B 0,C 180,E1 -23079.897,E2 -23079.897} C_VEL
LIN {X 0,Y 219.957,Z 585.189,A -85,B 0,C 180,E1 -23082.143,E2 -23082.143} C_VEL
LIN {X 0,Y 219.812,Z 585.854,A -85,B 0,C 180,E1 -23084.7,E2 -23084.7} C_VEL
LIN {X 0,Y 219.655,Z 586.152,A -85,B 0,C 180,E1 -23085.259,E2 -23085.259} C_VEL
LIN {X 0,Y 218.499,Z 587.239,A -85,B 0,C 180,E1 -23086.247,E2 -23086.247} C_VEL
LIN {X 0,Y 213.124,Z 591.432,A -85,B 0,C 180,E1 -23088.736,E2 -23088.736} C_VEL
LIN {X 0,Y 207.395,Z 595.581,A -85,B 0,C 180,E1 -23091.177,E2 -23091.177} C_VEL
LIN {X 0,Y 196.66,Z 601.796,A -85,B 0,C 180,E1 -23095.125,E2 -23095.125} C_VEL
LIN {X 0,Y 189.098,Z 605.472,A -85,B 0,C 180,E1 -23098.646,E2 -23098.646} C_VEL
LIN {X 0,Y 182.561,Z 608.018,A -85,B 0,C 180,E1 -23102.486,E2 -23102.486} C_VEL
LIN {X 0,Y 177.457,Z 609.445,A -85,B 0,C 180,E1 -23106.669,E2 -23106.669} C_VEL
LIN {X 0,Y 173.555,Z 609.732,A -85,B 0,C 180,E1 -23111.098,E2 -23111.098} C_VEL
LIN {X 0,Y 171.097,Z 608.876,A -85,B 0,C 180,E1 -23115.732,E2 -23115.732} C_VEL
LIN {X 0,Y 170.067,Z 606.838,A -85,B 0,C 180,E1 -23120.485,E2 -23120.485} C_VEL
LIN {X 0,Y 170.222,Z 603.454,A -85,B 0,C 180,E1 -23125.263,E2 -23125.263} C_VEL
LIN {X 0,Y 171.223,Z 599.347,A -85,B 0,C 180,E1 -23129.412,E2 -23129.412} C_VEL
LIN {X 0,Y 170.637,Z 602.739,A -85,B 0,C 180,E1 -23132.361,E2 -23132.361} C_VEL
LIN {X 0,Y 169.984,Z 606.723,A -85,B 0,C 180,E1 -23137.125,E2 -23137.125} C_VEL
LIN {X 0,Y 170.422,Z 609.334,A -85,B 0,C 180,E1 -23141.899,E2 -23141.899} C_VEL
LIN {X 0,Y 172.082,Z 610.7,A -85,B 0,C 180,E1 -23146.612,E2 -23146.612} C_VEL
LIN {X 0,Y 173.039,Z 610.879,A -85,B 0,C 180,E1 -23148.166,E2 -23148.166} C_VEL
LIN {X 0,Y 173.766,Z 610.948,A -85,B 0,C 180,E1 -23150.102,E2 -23150.102} C_VEL
LIN {X 0,Y 173.725,Z 610.531,A -85,B 0,C 180,E1 -23153.367,E2 -23153.367} C_VEL
LIN {X 0,Y 174.024,Z 609.904,A -85,B 0,C 180,E1 -23155.972,E2 -23155.972} C_VEL
LIN {X 0,Y 175.269,Z 609.373,A -85,B 0,C 180,E1 -23157.857,E2 -23157.857} C_VEL
LIN {X 0,Y 175.98,Z 609.143,A -85,B 0,C 180,E1 -23158.453,E2 -23158.453} C_VEL
LIN {X 0,Y 182.912,Z 606.976,A -85,B 0,C 180,E1 -23162.542,E2 -23162.542} C_VEL
LIN {X 0,Y 192.96,Z 602.797,A -85,B 0,C 180,E1 -23166.939,E2 -23166.939} C_VEL
LIN {X 0,Y 202.56,Z 597.866,A -85,B 0,C 180,E1 -23170.244,E2 -23170.244} C_VEL
LIN {X 0,Y 204.076,Z 596.946,A -85,B 0,C 180,E1 -23170.869,E2 -23170.869} C_VEL
LIN {X 0,Y 207.312,Z 594.629,A -85,B 0,C 180,E1 -23172.689,E2 -23172.689} C_VEL
LIN {X 0,Y 210.014,Z 592.597,A -85,B 0,C 180,E1 -23174.648,E2 -23174.648} C_VEL
LIN {X 0,Y 210.587,Z 592,A -85,B 0,C 180,E1 -23175.506,E2 -23175.506} C_VEL
LIN {X 0,Y 211.071,Z 591.34,A -85,B 0,C 180,E1 -23177.099,E2 -23177.099} C_VEL
LIN {X 0,Y 211.098,Z 591.115,A -85,B 0,C 180,E1 -23178.253,E2 -23178.253} C_VEL
LIN {X 0,Y 210.547,Z 591.186,A -85,B 0,C 180,E1 -23180.639,E2 -23180.639} C_VEL
LIN {X 0,Y 206.323,Z 593.101,A -85,B 0,C 180,E1 -23182.184,E2 -23182.184} C_VEL
LIN {X 0,Y 197.12,Z 596.659,A -85,B 0,C 180,E1 -23185.218,E2 -23185.218} C_VEL
LIN {X 0,Y 188.84,Z 598.961,A -85,B 0,C 180,E1 -23188.599,E2 -23188.599} C_VEL
LIN {X 0,Y 181.582,Z 600.083,A -85,B 0,C 180,E1 -23192.326,E2 -23192.326} C_VEL
LIN {X 0,Y 175.449,Z 600.034,A -85,B 0,C 180,E1 -23196.386,E2 -23196.386} C_VEL
LIN {X 0,Y 170.472,Z 598.778,A -85,B 0,C 180,E1 -23200.743,E2 -23200.743} C_VEL
LIN {X 0,Y 166.644,Z 596.285,A -85,B 0,C 180,E1 -23205.343,E2 -23205.343} C_VEL
LIN {X 0,Y 164.158,Z 592.547,A -85,B 0,C 180,E1 -23210.14,E2 -23210.14} C_VEL
LIN {X 0,Y 162.997,Z 587.476,A -85,B 0,C 180,E1 -23215.054,E2 -23215.054} C_VEL
LIN {X 0,Y 162.561,Z 582.594,A -85,B 0,C 180,E1 -23218.762,E2 -23218.762} C_VEL
LIN {X 0,Y 162.617,Z 575.603,A -85,B 0,C 180,E1 -23223.097,E2 -23223.097} C_VEL
LIN {X 0,Y 163.082,Z 566.885,A -85,B 0,C 180,E1 -23227.429,E2 -23227.429} C_VEL
LIN {X 0,Y 163.802,Z 557.631,A -85,B 0,C 180,E1 -23231.133,E2 -23231.133} C_VEL
LIN {X 0,Y 164.89,Z 547.395,A -85,B 0,C 180,E1 -23234.502,E2 -23234.502} C_VEL
LIN {X 0,Y 166.228,Z 536.203,A -85,B 0,C 180,E1 -23237.533,E2 -23237.533} C_VEL
LIN {X 0,Y 167.589,Z 525.604,A -85,B 0,C 180,E1 -23239.906,E2 -23239.906} C_VEL
LIN {X 0,Y 167.696,Z 522.554,A -85,B 0,C 180,E1 -23240.5,E2 -23240.5} C_VEL
LIN {X 0,Y 165.451,Z 510.143,A -85,B 0,C 180,E1 -23242.642,E2 -23242.642} C_VEL
LIN {X 0,Y 163.222,Z 496.153,A -85,B 0,C 180,E1 -23244.569,E2 -23244.569} C_VEL
LIN {X 0,Y 163.686,Z 496.092,A -85,B 0,C 180,E1 -23251.014,E2 -23251.014} C_VEL
LIN {X 0,Y 164.035,Z 496.05,A -85,B 0,C 180,E1 -23255.507,E2 -23255.507} C_VEL
LIN {X 0,Y 164.23,Z 496.027,A -85,B 0,C 180,E1 -23259.935,E2 -23259.935} C_VEL
LIN {X 0,Y 164.282,Z 496.018,A -85,B 0,C 180,E1 -23263.342,E2 -23263.342} C_VEL
LIN {X 0,Y 164.295,Z 496.019,A -85,B 0,C 180,E1 -23266.809,E2 -23266.809} C_VEL
LIN {X 0,Y 164.308,Z 496.013,A -85,B 0,C 180,E1 -23270.348,E2 -23270.348} C_VEL
LIN {X 0,Y 164.347,Z 496.014,A -85,B 0,C 180,E1 -23274.343,E2 -23274.343} C_VEL
LIN {X 0,Y 164.395,Z 496,A -85,B 0,C 180,E1 -23279.135,E2 -23279.135} C_VEL
LIN {X 0,Y 164.42,Z 496.003,A -85,B 0,C 180,E1 -23284.695,E2 -23284.695} C_VEL
LIN {X 0,Y 164.488,Z 495.994,A -85,B 0,C 180,E1 -23290.051,E2 -23290.051} C_VEL
LIN {X 0,Y 164.558,Z 495.984,A -85,B 0,C 180,E1 -23295.152,E2 -23295.152} C_VEL
LIN {X 0,Y 164.857,Z 495.951,A -85,B 0,C 180,E1 -23300.182,E2 -23300.182} C_VEL
LIN {X 0,Y 164.867,Z 495.947,A -85,B 0,C 180,E1 -23302.653,E2 -23302.653} C_VEL
LIN {X 0,Y 165.055,Z 495.922,A -85,B 0,C 180,E1 -23307.56,E2 -23307.56} C_VEL
LIN {X 0,Y 165.299,Z 495.896,A -85,B 0,C 180,E1 -23310,E2 -23310} C_VEL
LIN {X 0,Y 164.762,Z 495.956,A -85,B 0,C 180,E1 -23314.894,E2 -23314.894} C_VEL
LIN {X 0,Y 164.831,Z 495.951,A -85,B 0,C 180,E1 -23317.349,E2 -23317.349} C_VEL
LIN {X 0,Y 164.706,Z 495.966,A -85,B 0,C 180,E1 -23321.061,E2 -23321.061} C_VEL
LIN {X 0,Y 164.488,Z 495.995,A -85,B 0,C 180,E1 -23327.403,E2 -23327.403} C_VEL
LIN {X 0,Y 164.477,Z 495.995,A -85,B 0,C 180,E1 -23329.989,E2 -23329.989} C_VEL
LIN {X 0,Y 164.397,Z 496.007,A -85,B 0,C 180,E1 -23336.134,E2 -23336.134} C_VEL
LIN {X 0,Y 164.379,Z 496.002,A -85,B 0,C 180,E1 -23341.228,E2 -23341.228} C_VEL
LIN {X 0,Y 164.316,Z 496.015,A -85,B 0,C 180,E1 -23346.784,E2 -23346.784} C_VEL
LIN {X 0,Y 164.303,Z 496.014,A -85,B 0,C 180,E1 -23349.913,E2 -23349.913} C_VEL
LIN {X 0,Y 164.282,Z 496.021,A -85,B 0,C 180,E1 -23353.341,E2 -23353.341} C_VEL
LIN {X 0,Y 164.295,Z 496.016,A -85,B 0,C 180,E1 -23356.808,E2 -23356.808} C_VEL
LIN {X 0,Y 164.262,Z 496.022,A -85,B 0,C 180,E1 -23360.367,E2 -23360.367} C_VEL
LIN {X 0,Y 164.142,Z 496.036,A -85,B 0,C 180,E1 -23364.441,E2 -23364.441} C_VEL
LIN {X 0,Y 163.756,Z 496.084,A -85,B 0,C 180,E1 -23369.132,E2 -23369.132} C_VEL
LIN {X 0,Y 163.271,Z 496.143,A -85,B 0,C 180,E1 -23374.682,E2 -23374.682} C_VEL
LIN {X 0,Y 163.234,Z 496.253,A -85,B 0,C 180,E1 -23375.896,E2 -23375.896} C_VEL
LIN {X 0,Y 165.663,Z 511.163,A -85,B 0,C 180,E1 -23377.979,E2 -23377.979} C_VEL
LIN {X 0,Y 167.597,Z 522,A -85,B 0,C 180,E1 -23379.852,E2 -23379.852} C_VEL
LIN {X 0,Y 167.188,Z 527.632,A -85,B 0,C 180,E1 -23380.986,E2 -23380.986} C_VEL
LIN {X 0,Y 165.591,Z 540.28,A -85,B 0,C 180,E1 -23383.985,E2 -23383.985} C_VEL
LIN {X 0,Y 164.252,Z 552.585,A -85,B 0,C 180,E1 -23387.646,E2 -23387.646} C_VEL
LIN {X 0,Y 163.249,Z 562.61,A -85,B 0,C 180,E1 -23391.334,E2 -23391.334} C_VEL
LIN {X 0,Y 162.689,Z 570.825,A -85,B 0,C 180,E1 -23395.043,E2 -23395.043} C_VEL
LIN {X 0,Y 162.561,Z 577.658,A -85,B 0,C 180,E1 -23398.761,E2 -23398.761} C_VEL
LIN {X 0,Y 162.643,Z 583.292,A -85,B 0,C 180,E1 -23402.476,E2 -23402.476} C_VEL
LIN {X 0,Y 163.155,Z 587.874,A -85,B 0,C 180,E1 -23406.182,E2 -23406.182} C_VEL
LIN {X 0,Y 164.558,Z 592.697,A -85,B 0,C 180,E1 -23411.08,E2 -23411.08} C_VEL
LIN {X 0,Y 166.555,Z 595.386,A -85,B 0,C 180,E1 -23414.665,E2 -23414.665} C_VEL
LIN {X 0,Y 170.163,Z 597.906,A -85,B 0,C 180,E1 -23419.293,E2 -23419.293} C_VEL
LIN {X 0,Y 175.282,Z 599.199,A -85,B 0,C 180,E1 -23423.637,E2 -23423.637} C_VEL
LIN {X 0,Y 181.359,Z 599.265,A -85,B 0,C 180,E1 -23427.711,E2 -23427.711} C_VEL
LIN {X 0,Y 188.637,Z 598.13,A -85,B 0,C 180,E1 -23431.439,E2 -23431.439} C_VEL
LIN {X 0,Y 197.611,Z 595.569,A -85,B 0,C 180,E1 -23435.116,E2 -23435.116} C_VEL
LIN {X 0,Y 206.008,Z 592.257,A -85,B 0,C 180,E1 -23437.884,E2 -23437.884} C_VEL
LIN {X 0,Y 210.904,Z 590.003,A -85,B 0,C 180,E1 -23439.282,E2 -23439.282} C_VEL
LIN {X 0,Y 212.914,Z 588.974,A -85,B 0,C 180,E1 -23440.059,E2 -23440.059} C_VEL
LIN {X 0,Y 213.336,Z 588.808,A -85,B 0,C 180,E1 -23441.213,E2 -23441.213} C_VEL
LIN {X 0,Y 213.71,Z 589.052,A -85,B 0,C 180,E1 -23443.677,E2 -23443.677} C_VEL
LIN {X 0,Y 213.388,Z 589.604,A -85,B 0,C 180,E1 -23444.928,E2 -23444.928} C_VEL
LIN {X 0,Y 211.824,Z 590.719,A -85,B 0,C 180,E1 -23445.833,E2 -23445.833} C_VEL
LIN {X 0,Y 204.118,Z 595.804,A -85,B 0,C 180,E1 -23449.142,E2 -23449.142} C_VEL
LIN {X 0,Y 198.776,Z 598.813,A -85,B 0,C 180,E1 -23451.063,E2 -23451.063} C_VEL
LIN {X 0,Y 190.925,Z 602.611,A -85,B 0,C 180,E1 -23453.916,E2 -23453.916} C_VEL
LIN {X 0,Y 183.096,Z 605.824,A -85,B 0,C 180,E1 -23457.494,E2 -23457.494} C_VEL
LIN {X 0,Y 176.285,Z 607.945,A -85,B 0,C 180,E1 -23461.419,E2 -23461.419} C_VEL
LIN {X 0,Y 170.96,Z 608.975,A -85,B 0,C 180,E1 -23465.727,E2 -23465.727} C_VEL
LIN {X 0,Y 166.877,Z 608.899,A -85,B 0,C 180,E1 -23470.311,E2 -23470.311} C_VEL
LIN {X 0,Y 164.283,Z 607.717,A -85,B 0,C 180,E1 -23475.127,E2 -23475.127} C_VEL
LIN {X 0,Y 163.186,Z 605.373,A -85,B 0,C 180,E1 -23480.08,E2 -23480.08} C_VEL
LIN {X 0,Y 163.359,Z 601.744,A -85,B 0,C 180,E1 -23485.064,E2 -23485.064} C_VEL
LIN {X 0,Y 164.416,Z 597.398,A -85,B 0,C 180,E1 -23489.464,E2 -23489.464} C_VEL
LIN {X 0,Y 163.787,Z 600.864,A -85,B 0,C 180,E1 -23492.459,E2 -23492.459} C_VEL
LIN {X 0,Y 163.106,Z 605.324,A -85,B 0,C 180,E1 -23497.679,E2 -23497.679} C_VEL
LIN {X 0,Y 163.566,Z 608.014,A -85,B 0,C 180,E1 -23502.406,E2 -23502.406} C_VEL
LIN {X 0,Y 165.333,Z 609.695,A -85,B 0,C 180,E1 -23507.311,E2 -23507.311} C_VEL
LIN {X 0,Y 168.749,Z 610.287,A -85,B 0,C 180,E1 -23512.014,E2 -23512.014} C_VEL
LIN {X 0,Y 173.422,Z 609.766,A -85,B 0,C 180,E1 -23516.473,E2 -23516.473} C_VEL
LIN {X 0,Y 175.98,Z 609.143,A -85,B 0,C 180,E1 -23518.453,E2 -23518.453} C_VEL
LIN {X 0,Y 177.92,Z 608.522,A -85,B 0,C 180,E1 -23520.253,E2 -23520.253} C_VEL
LIN {X 0,Y 182.342,Z 605.802,A -85,B 0,C 180,E1 -23525.674,E2 -23525.674} C_VEL
LIN {X 0,Y 184.949,Z 604.523,A -85,B 0,C 180,E1 -23527.264,E2 -23527.264} C_VEL
LIN {X 0,Y 186.077,Z 604.051,A -85,B 0,C 180,E1 -23527.735,E2 -23527.735} C_VEL
LIN {X 0,Y 194.4,Z 600.578,A -85,B 0,C 180,E1 -23530.598,E2 -23530.598} C_VEL
LIN {X 0,Y 197.622,Z 598.999,A -85,B 0,C 180,E1 -23531.685,E2 -23531.685} C_VEL
LIN {X 0,Y 200.527,Z 597.325,A -85,B 0,C 180,E1 -23533.112,E2 -23533.112} C_VEL
LIN {X 0,Y 202.125,Z 596.329,A -85,B 0,C 180,E1 -23534.06,E2 -23534.06} C_VEL
LIN {X 0,Y 204.323,Z 594.707,A -85,B 0,C 180,E1 -23536.247,E2 -23536.247} C_VEL
LIN {X 0,Y 204.398,Z 594.082,A -85,B 0,C 180,E1 -23539.21,E2 -23539.21} C_VEL
LIN {X 0,Y 200.987,Z 595.346,A -85,B 0,C 180,E1 -23540.993,E2 -23540.993} C_VEL
LIN {X 0,Y 191.485,Z 598.366,A -85,B 0,C 180,E1 -23544.039,E2 -23544.039} C_VEL
LIN {X 0,Y 182.906,Z 600.207,A -85,B 0,C 180,E1 -23547.457,E2 -23547.457} C_VEL
LIN {X 0,Y 175.375,Z 600.887,A -85,B 0,C 180,E1 -23551.257,E2 -23551.257} C_VEL
LIN {X 0,Y 169.001,Z 600.407,A -85,B 0,C 180,E1 -23555.427,E2 -23555.427} C_VEL
LIN {X 0,Y 163.81,Z 598.766,A -85,B 0,C 180,E1 -23559.927,E2 -23559.927} C_VEL
LIN {X 0,Y 159.808,Z 595.938,A -85,B 0,C 180,E1 -23564.701,E2 -23564.701} C_VEL
LIN {X 0,Y 157.219,Z 591.848,A -85,B 0,C 180,E1 -23569.7,E2 -23569.7} C_VEL
LIN {X 0,Y 156.022,Z 586.378,A -85,B 0,C 180,E1 -23574.832,E2 -23574.832} C_VEL
LIN {X 0,Y 155.537,Z 579.333,A -85,B 0,C 180,E1 -23580.001,E2 -23580.001} C_VEL
LIN {X 0,Y 155.668,Z 572.685,A -85,B 0,C 180,E1 -23583.884,E2 -23583.884} C_VEL
LIN {X 0,Y 156.218,Z 563.632,A -85,B 0,C 180,E1 -23588.211,E2 -23588.211} C_VEL
LIN {X 0,Y 157.175,Z 553.278,A -85,B 0,C 180,E1 -23592.263,E2 -23592.263} C_VEL
LIN {X 0,Y 158.431,Z 542.057,A -85,B 0,C 180,E1 -23595.767,E2 -23595.767} C_VEL
LIN {X 0,Y 159.984,Z 529.695,A -85,B 0,C 180,E1 -23598.905,E2 -23598.905} C_VEL
LIN {X 0,Y 160.641,Z 523.868,A -85,B 0,C 180,E1 -23600.154,E2 -23600.154} C_VEL
LIN {X 0,Y 158.429,Z 511.026,A -85,B 0,C 180,E1 -23602.493,E2 -23602.493} C_VEL
LIN {X 0,Y 156.195,Z 497.028,A -85,B 0,C 180,E1 -23604.548,E2 -23604.548} C_VEL
LIN {X 0,Y 156.668,Z 496.966,A -85,B 0,C 180,E1 -23611.534,E2 -23611.534} C_VEL
LIN {X 0,Y 157.02,Z 496.926,A -85,B 0,C 180,E1 -23616.326,E2 -23616.326} C_VEL
LIN {X 0,Y 157.152,Z 496.905,A -85,B 0,C 180,E1 -23620.513,E2 -23620.513} C_VEL
LIN {X 0,Y 157.18,Z 496.905,A -85,B 0,C 180,E1 -23625.678,E2 -23625.678} C_VEL
LIN {X 0,Y 157.241,Z 496.893,A -85,B 0,C 180,E1 -23631.263,E2 -23631.263} C_VEL
LIN {X 0,Y 157.294,Z 496.892,A -85,B 0,C 180,E1 -23634.49,E2 -23634.49} C_VEL
LIN {X 0,Y 157.298,Z 496.887,A -85,B 0,C 180,E1 -23638.095,E2 -23638.095} C_VEL
LIN {X 0,Y 157.326,Z 496.887,A -85,B 0,C 180,E1 -23643.467,E2 -23643.467} C_VEL
LIN {X 0,Y 157.398,Z 496.875,A -85,B 0,C 180,E1 -23649.668,E2 -23649.668} C_VEL
LIN {X 0,Y 157.483,Z 496.866,A -85,B 0,C 180,E1 -23654.469,E2 -23654.469} C_VEL
LIN {X 0,Y 157.777,Z 496.83,A -85,B 0,C 180,E1 -23659.736,E2 -23659.736} C_VEL
LIN {X 0,Y 157.829,Z 496.824,A -85,B 0,C 180,E1 -23662.323,E2 -23662.323} C_VEL
LIN {X 0,Y 158.261,Z 496.773,A -85,B 0,C 180,E1 -23670,E2 -23670} C_VEL
LIN {X 0,Y 157.768,Z 496.832,A -85,B 0,C 180,E1 -23677.68,E2 -23677.68} C_VEL
LIN {X 0,Y 157.641,Z 496.846,A -85,B 0,C 180,E1 -23681.237,E2 -23681.237} C_VEL
LIN {X 0,Y 157.458,Z 496.869,A -85,B 0,C 180,E1 -23685.534,E2 -23685.534} C_VEL
LIN {X 0,Y 157.374,Z 496.877,A -85,B 0,C 180,E1 -23690.932,E2 -23690.932} C_VEL
LIN {X 0,Y 157.318,Z 496.888,A -85,B 0,C 180,E1 -23696.685,E2 -23696.685} C_VEL
LIN {X 0,Y 157.282,Z 496.891,A -85,B 0,C 180,E1 -23702.426,E2 -23702.426} C_VEL
LIN {X 0,Y 157.286,Z 496.891,A -85,B 0,C 180,E1 -23706.456,E2 -23706.456} C_VEL
LIN {X 0,Y 157.216,Z 496.901,A -85,B 0,C 180,E1 -23712.109,E2 -23712.109} C_VEL
LIN {X 0,Y 157.204,Z 496.897,A -85,B 0,C 180,E1 -23717.886,E2 -23717.886} C_VEL
LIN {X 0,Y 157.137,Z 496.912,A -85,B 0,C 180,E1 -23723.616,E2 -23723.616} C_VEL
LIN {X 0,Y 156.752,Z 496.956,A -85,B 0,C 180,E1 -23728.416,E2 -23728.416} C_VEL
LIN {X 0,Y 156.193,Z 497.025,A -85,B 0,C 180,E1 -23735.524,E2 -23735.524} C_VEL
LIN {X 0,Y 156.221,Z 497.19,A -85,B 0,C 180,E1 -23735.969,E2 -23735.969} C_VEL
LIN {X 0,Y 158.469,Z 510.836,A -85,B 0,C 180,E1 -23737.963,E2 -23737.963} C_VEL
LIN {X 0,Y 160.552,Z 523.056,A -85,B 0,C 180,E1 -23740.168,E2 -23740.168} C_VEL
LIN {X 0,Y 158.947,Z 536.709,A -85,B 0,C 180,E1 -23743.297,E2 -23743.297} C_VEL
LIN {X 0,Y 157.51,Z 548.764,A -85,B 0,C 180,E1 -23746.78,E2 -23746.78} C_VEL
LIN {X 0,Y 156.484,Z 558.763,A -85,B 0,C 180,E1 -23750.369,E2 -23750.369} C_VEL
LIN {X 0,Y 155.843,Z 567.233,A -85,B 0,C 180,E1 -23754.037,E2 -23754.037} C_VEL
LIN {X 0,Y 155.61,Z 574.984,A -85,B 0,C 180,E1 -23758.058,E2 -23758.058} C_VEL
LIN {X 0,Y 155.665,Z 581.987,A -85,B 0,C 180,E1 -23762.587,E2 -23762.587} C_VEL
LIN {X 0,Y 156.189,Z 586.889,A -85,B 0,C 180,E1 -23766.458,E2 -23766.458} C_VEL
LIN {X 0,Y 157.651,Z 592.015,A -85,B 0,C 180,E1 -23771.572,E2 -23771.572} C_VEL
LIN {X 0,Y 159.717,Z 595.018,A -85,B 0,C 180,E1 -23775.308,E2 -23775.308} C_VEL
LIN {X 0,Y 163.494,Z 597.887,A -85,B 0,C 180,E1 -23780.114,E2 -23780.114} C_VEL
LIN {X 0,Y 168.821,Z 599.547,A -85,B 0,C 180,E1 -23784.601,E2 -23784.601} C_VEL
LIN {X 0,Y 175.141,Z 600.037,A -85,B 0,C 180,E1 -23788.785,E2 -23788.785} C_VEL
LIN {X 0,Y 182.717,Z 599.347,A -85,B 0,C 180,E1 -23792.581,E2 -23792.581} C_VEL
LIN {X 0,Y 191.218,Z 597.523,A -85,B 0,C 180,E1 -23796.019,E2 -23796.019} C_VEL
LIN {X 0,Y 200.662,Z 594.496,A -85,B 0,C 180,E1 -23799.082,E2 -23799.082} C_VEL
LIN {X 0,Y 205.693,Z 592.477,A -85,B 0,C 180,E1 -23800.48,E2 -23800.48} C_VEL
LIN {X 0,Y 207.033,Z 591.997,A -85,B 0,C 180,E1 -23801.684,E2 -23801.684} C_VEL
LIN {X 0,Y 207.173,Z 592.117,A -85,B 0,C 180,E1 -23802.724,E2 -23802.724} C_VEL
LIN {X 0,Y 206.856,Z 592.689,A -85,B 0,C 180,E1 -23804.481,E2 -23804.481} C_VEL
LIN {X 0,Y 202.965,Z 594.982,A -85,B 0,C 180,E1 -23806.169,E2 -23806.169} C_VEL
LIN {X 0,Y 197.393,Z 598.02,A -85,B 0,C 180,E1 -23808.39,E2 -23808.39} C_VEL
LIN {X 0,Y 189.757,Z 601.526,A -85,B 0,C 180,E1 -23810.977,E2 -23810.977} C_VEL
LIN {X 0,Y 181.036,Z 604.812,A -85,B 0,C 180,E1 -23814.386,E2 -23814.386} C_VEL
LIN {X 0,Y 173.412,Z 607.039,A -85,B 0,C 180,E1 -23818.206,E2 -23818.206} C_VEL
LIN {X 0,Y 167.17,Z 608.208,A -85,B 0,C 180,E1 -23822.455,E2 -23822.455} C_VEL
LIN {X 0,Y 162.259,Z 608.316,A -85,B 0,C 180,E1 -23827.057,E2 -23827.057} C_VEL
LIN {X 0,Y 158.617,Z 607.33,A -85,B 0,C 180,E1 -23831.931,E2 -23831.931} C_VEL
LIN {X 0,Y 156.749,Z 605.271,A -85,B 0,C 180,E1 -23837.045,E2 -23837.045} C_VEL
LIN {X 0,Y 156.3,Z 601.999,A -85,B 0,C 180,E1 -23842.247,E2 -23842.247} C_VEL
LIN {X 0,Y 157.071,Z 597.354,A -85,B 0,C 180,E1 -23847.435,E2 -23847.435} C_VEL
LIN {X 0,Y 157.662,Z 595.21,A -85,B 0,C 180,E1 -23849.441,E2 -23849.441} C_VEL
LIN {X 0,Y 156.99,Z 598.858,A -85,B 0,C 180,E1 -23852.566,E2 -23852.566} C_VEL
LIN {X 0,Y 156.281,Z 603.42,A -85,B 0,C 180,E1 -23857.754,E2 -23857.754} C_VEL
LIN {X 0,Y 156.752,Z 606.626,A -85,B 0,C 180,E1 -23862.954,E2 -23862.954} C_VEL
LIN {X 0,Y 158.635,Z 608.591,A -85,B 0,C 180,E1 -23868.067,E2 -23868.067} C_VEL
LIN {X 0,Y 162.206,Z 609.517,A -85,B 0,C 180,E1 -23872.951,E2 -23872.951} C_VEL
LIN {X 0,Y 167.099,Z 609.365,A -85,B 0,C 180,E1 -23877.558,E2 -23877.558} C_VEL
LIN {X 0,Y 173.313,Z 608.164,A -85,B 0,C 180,E1 -23881.814,E2 -23881.814} C_VEL
LIN {X 0,Y 180.929,Z 605.933,A -85,B 0,C 180,E1 -23885.638,E2 -23885.638} C_VEL
LIN {X 0,Y 186.077,Z 604.051,A -85,B 0,C 180,E1 -23887.735,E2 -23887.735} C_VEL
LIN {X 0,Y 188.056,Z 603.152,A -85,B 0,C 180,E1 -23888.743,E2 -23888.743} C_VEL
LIN {X 0,Y 190.039,Z 601.862,A -85,B 0,C 180,E1 -23890.628,E2 -23890.628} C_VEL
LIN {X 0,Y 192.364,Z 600.257,A -85,B 0,C 180,E1 -23892.916,E2 -23892.916} C_VEL
LIN {X 0,Y 193.601,Z 599.632,A -85,B 0,C 180,E1 -23893.603,E2 -23893.603} C_VEL
LIN {X 0,Y 196.66,Z 597.911,A -85,B 0,C 180,E1 -23895.622,E2 -23895.622} C_VEL
LIN {X 0,Y 197.777,Z 597.039,A -85,B 0,C 180,E1 -23897.533,E2 -23897.533} C_VEL
LIN {X 0,Y 197.774,Z 596.892,A -85,B 0,C 180,E1 -23898.267,E2 -23898.267} C_VEL
